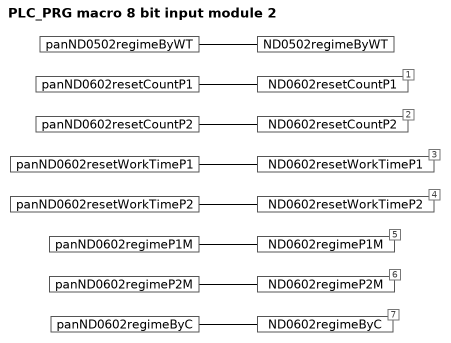
[picture p72: PLC_PRG macro 8 bit input module 2 (CFC)]
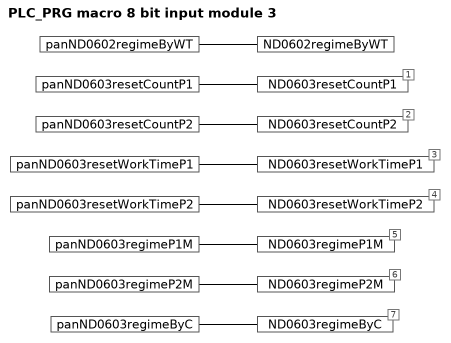
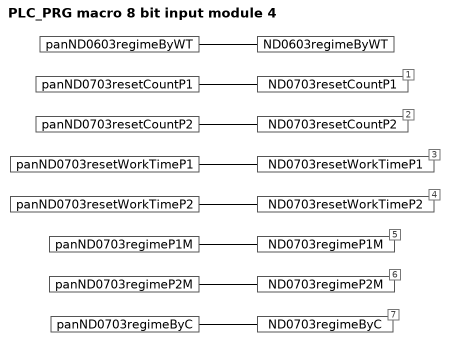
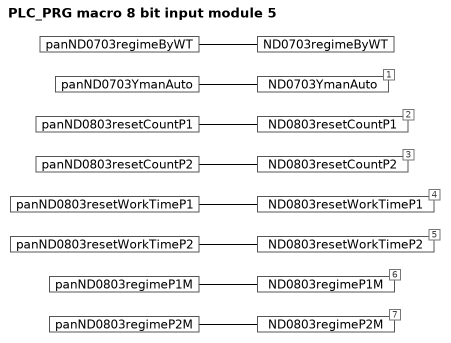
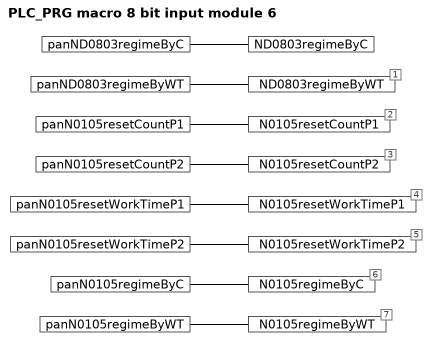
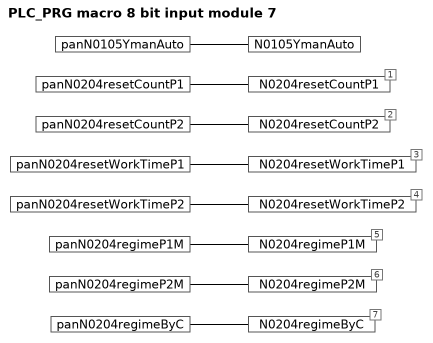
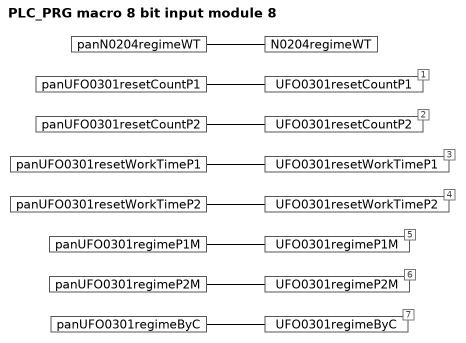
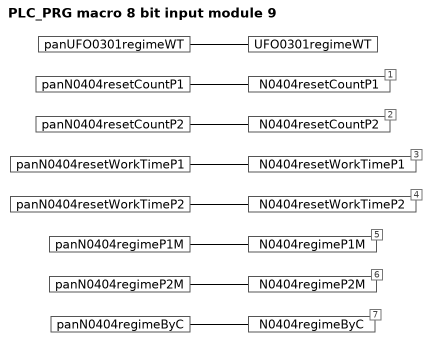
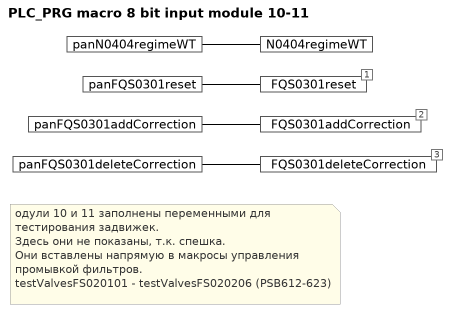
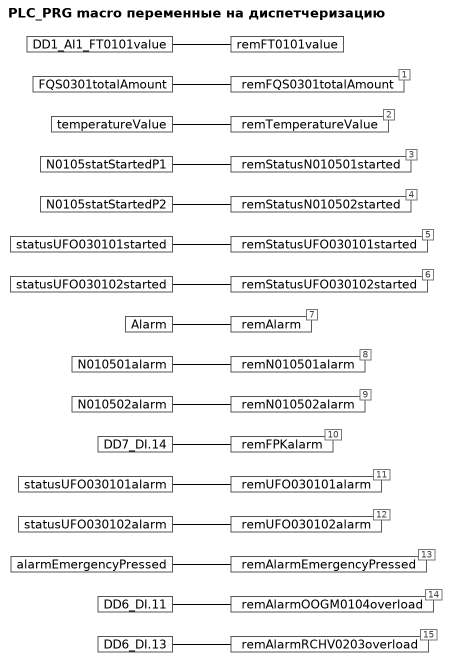
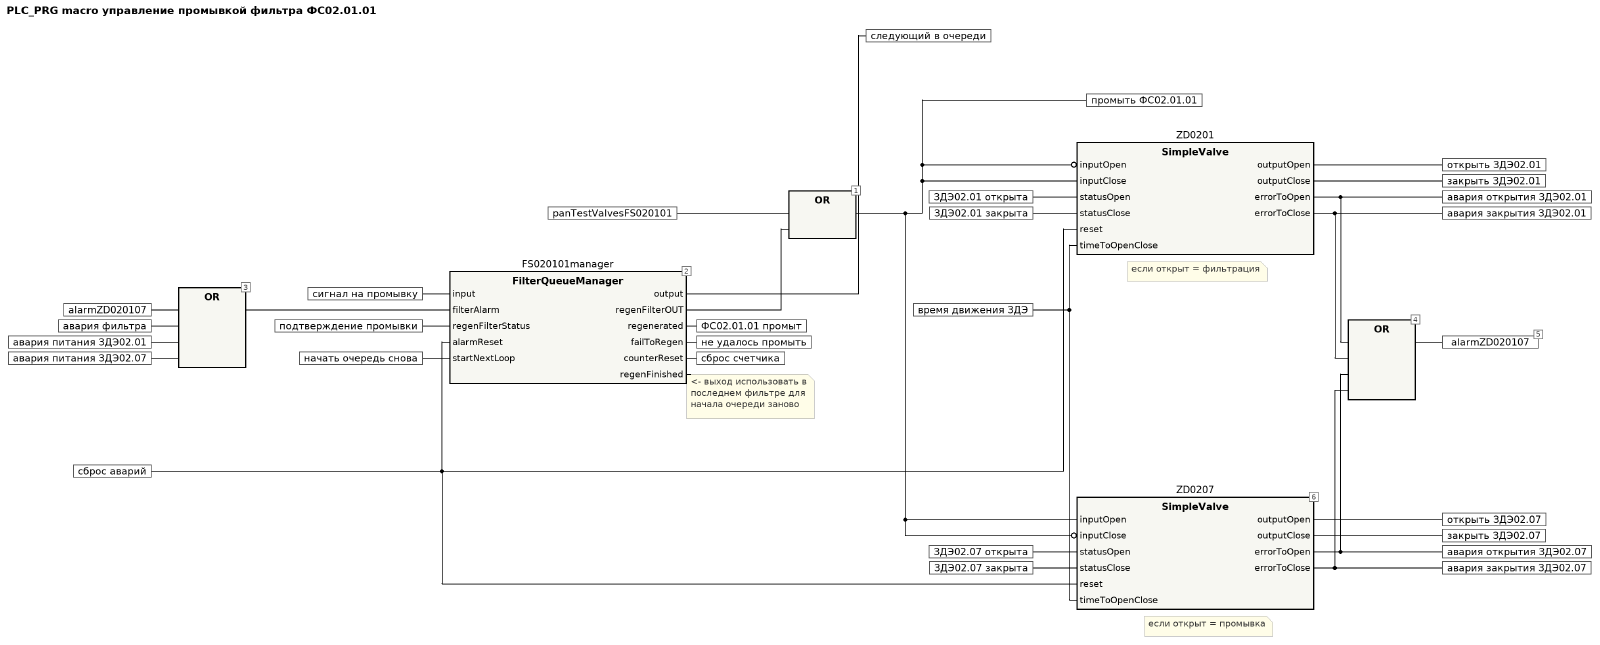
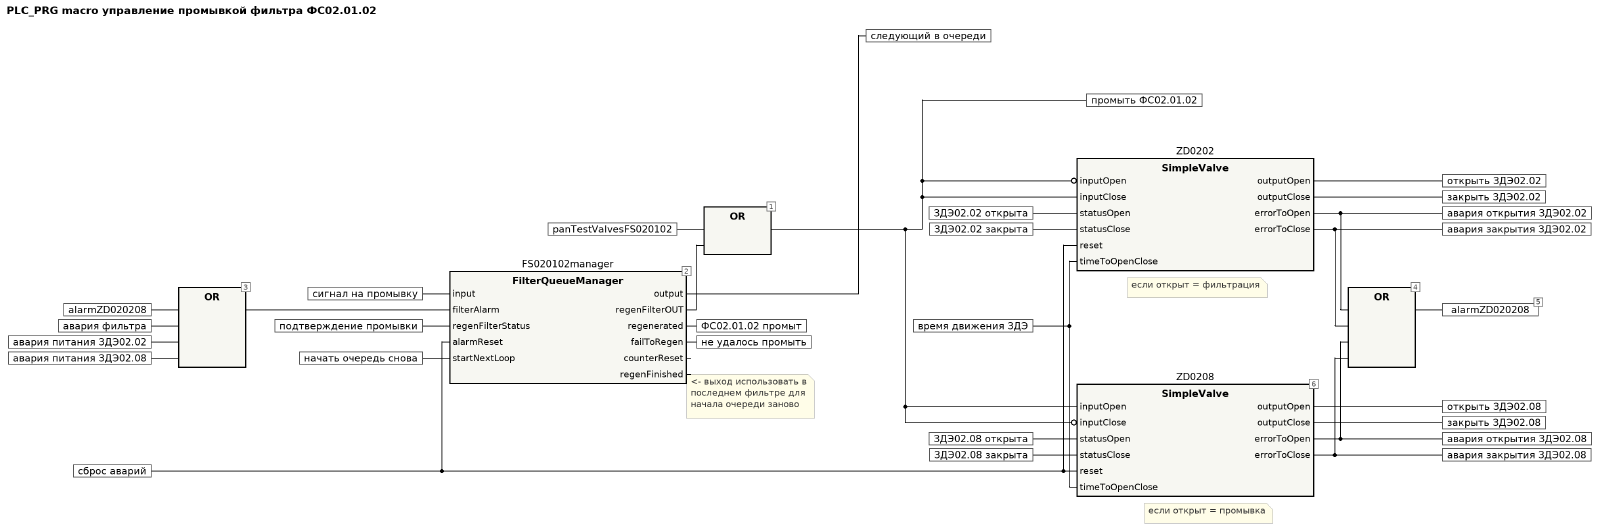
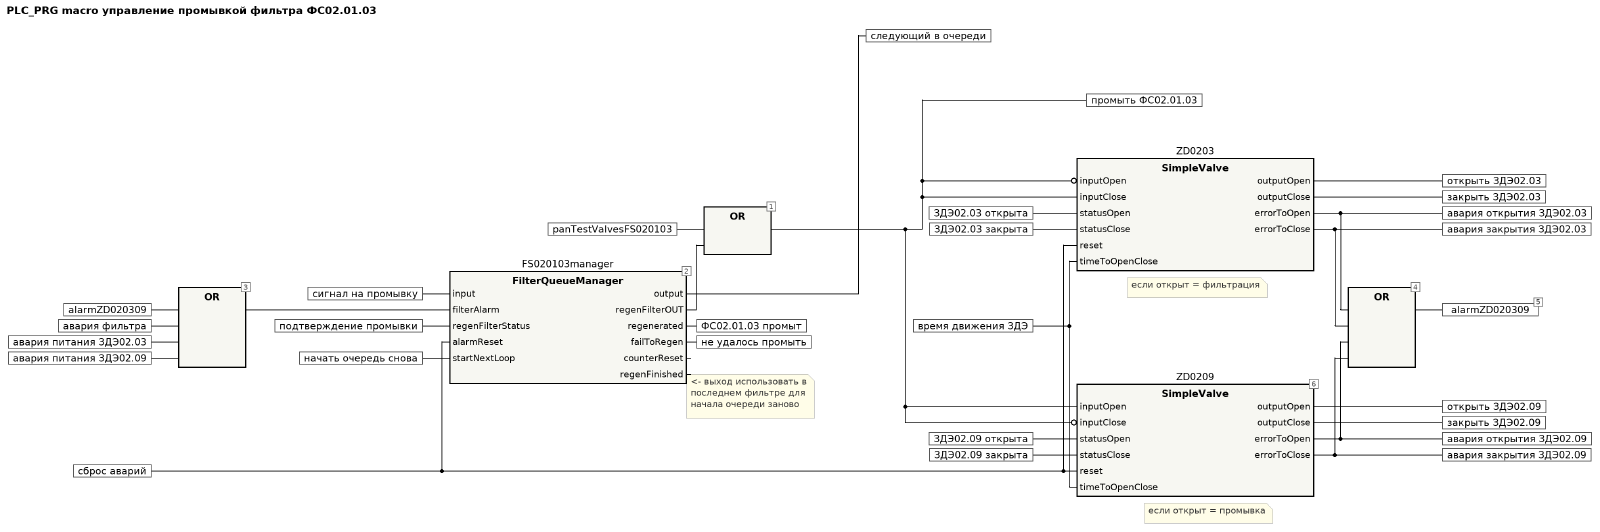
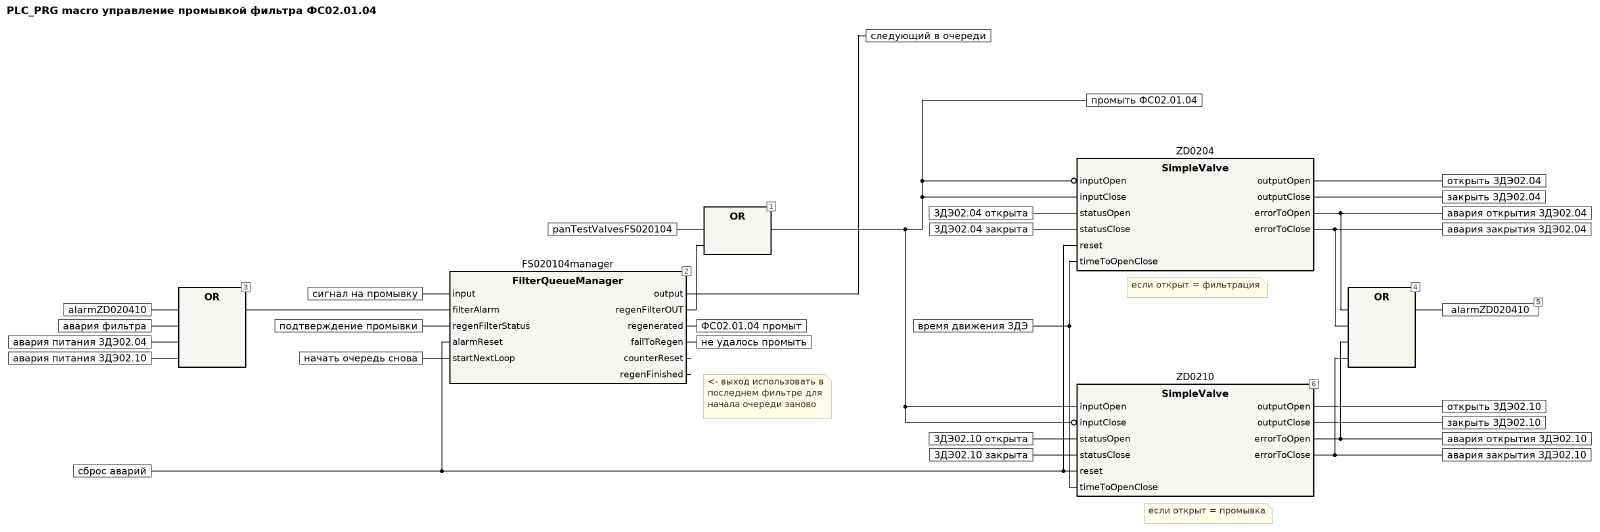
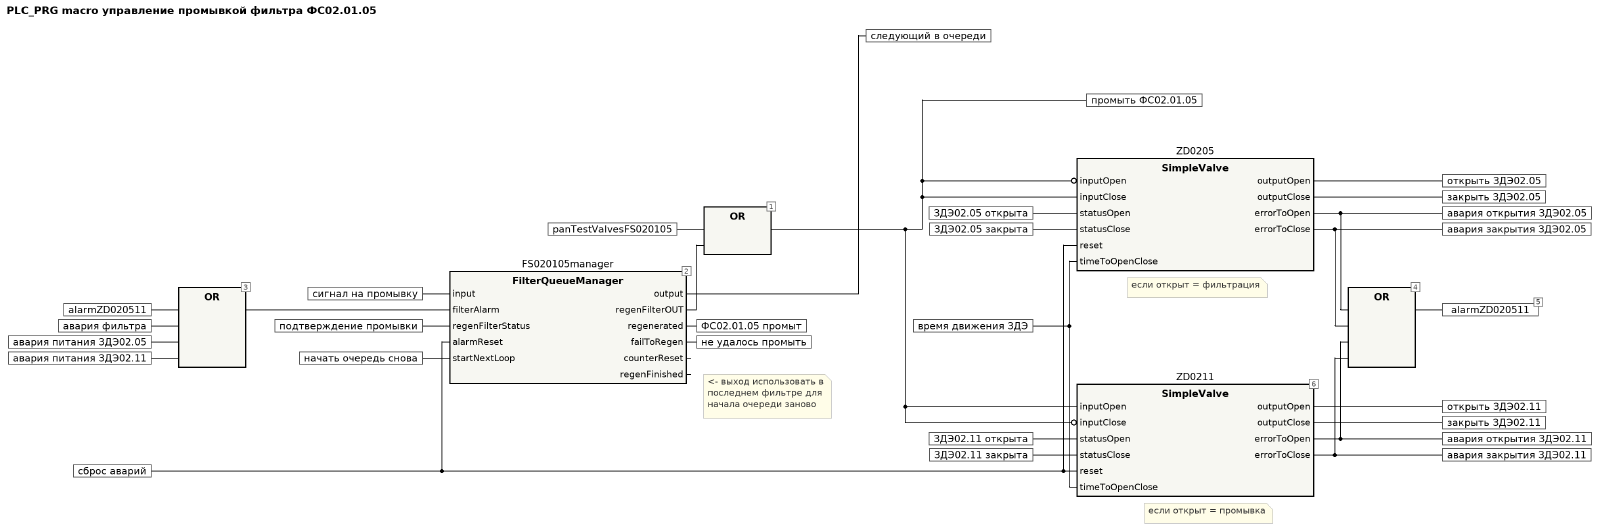
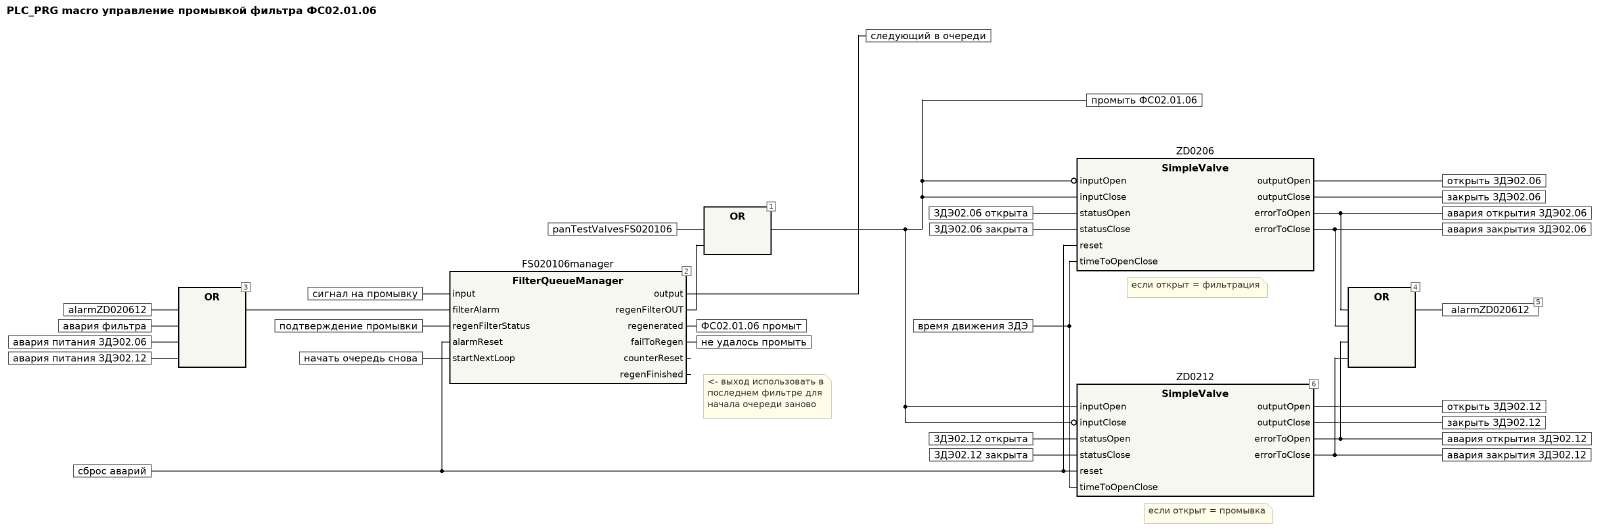
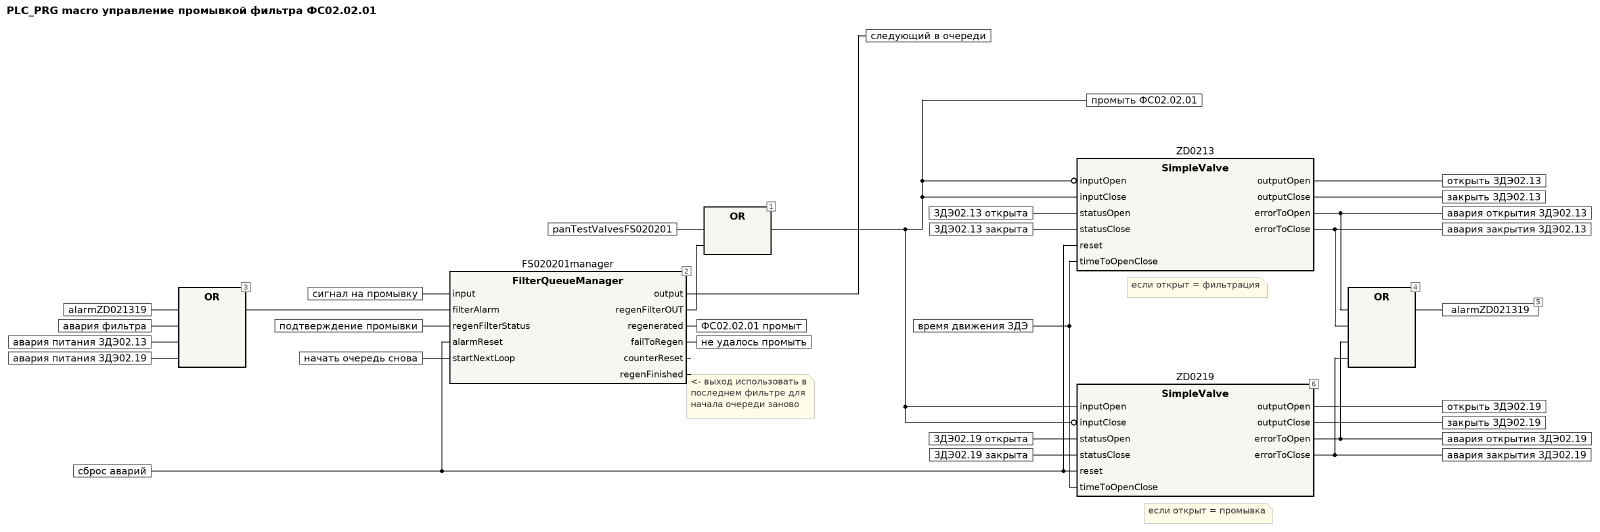
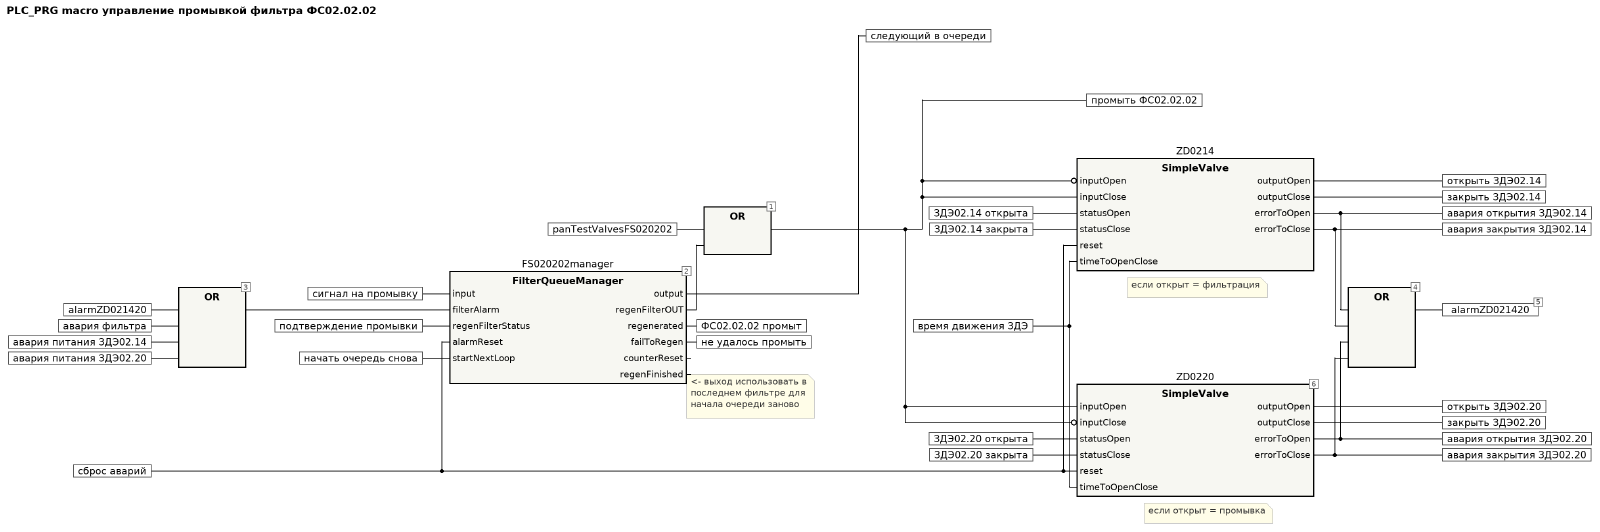
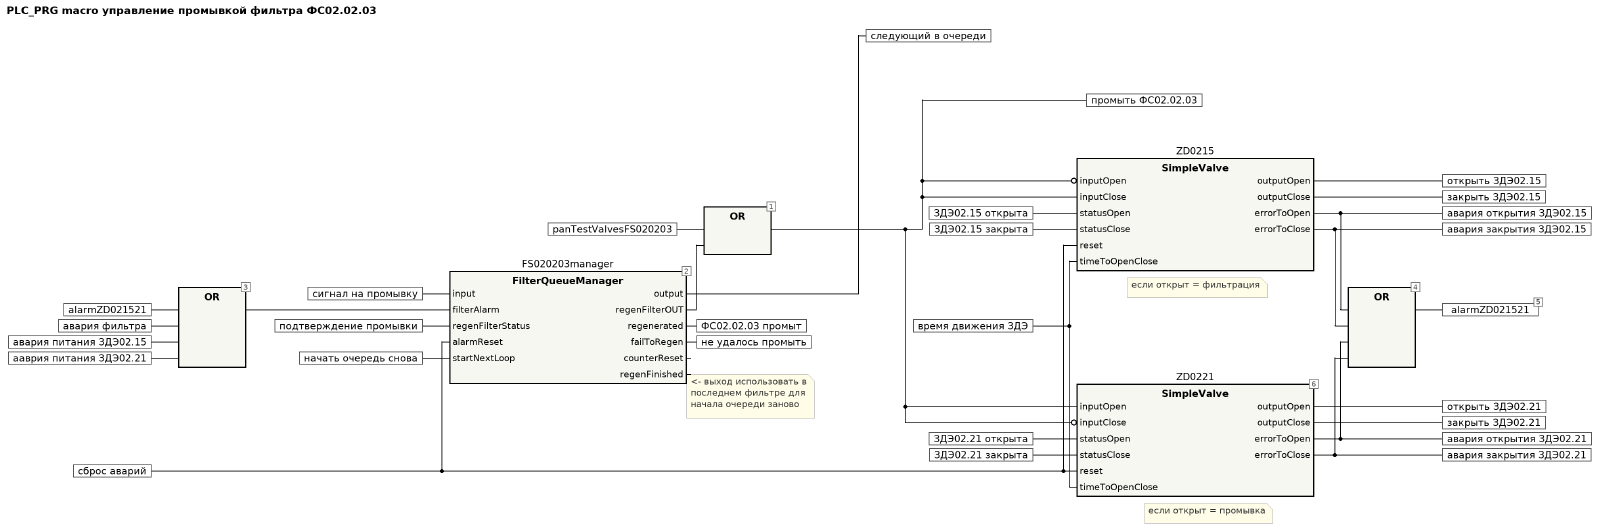
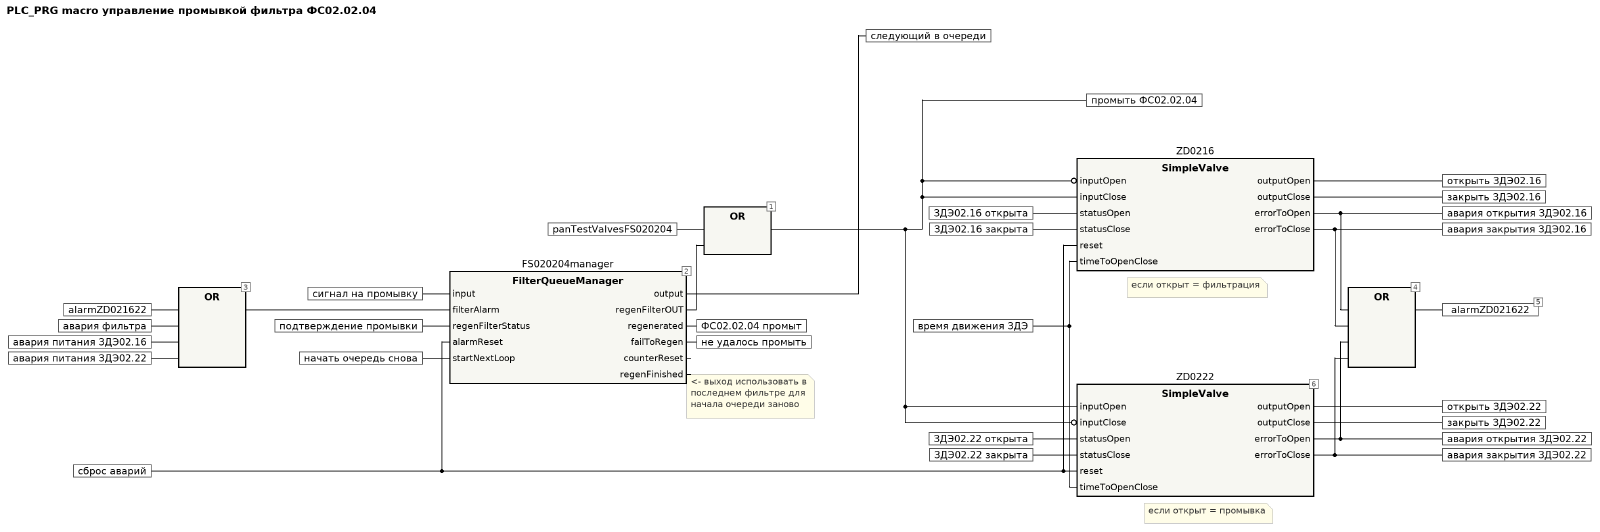
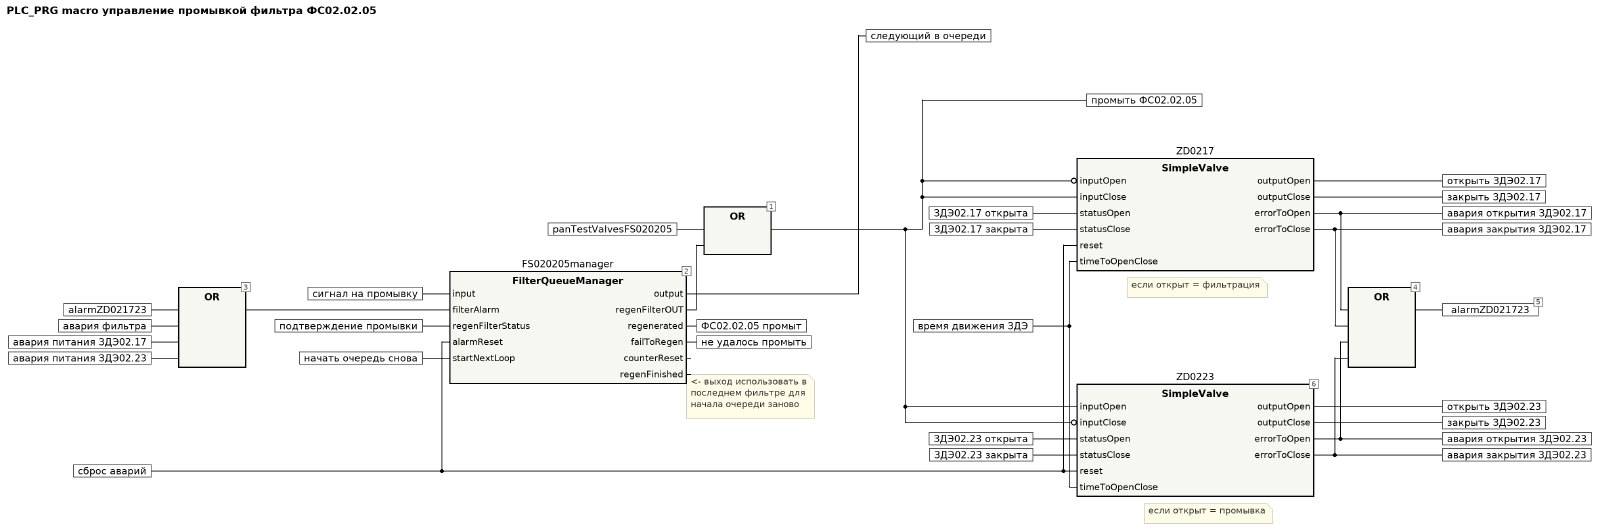
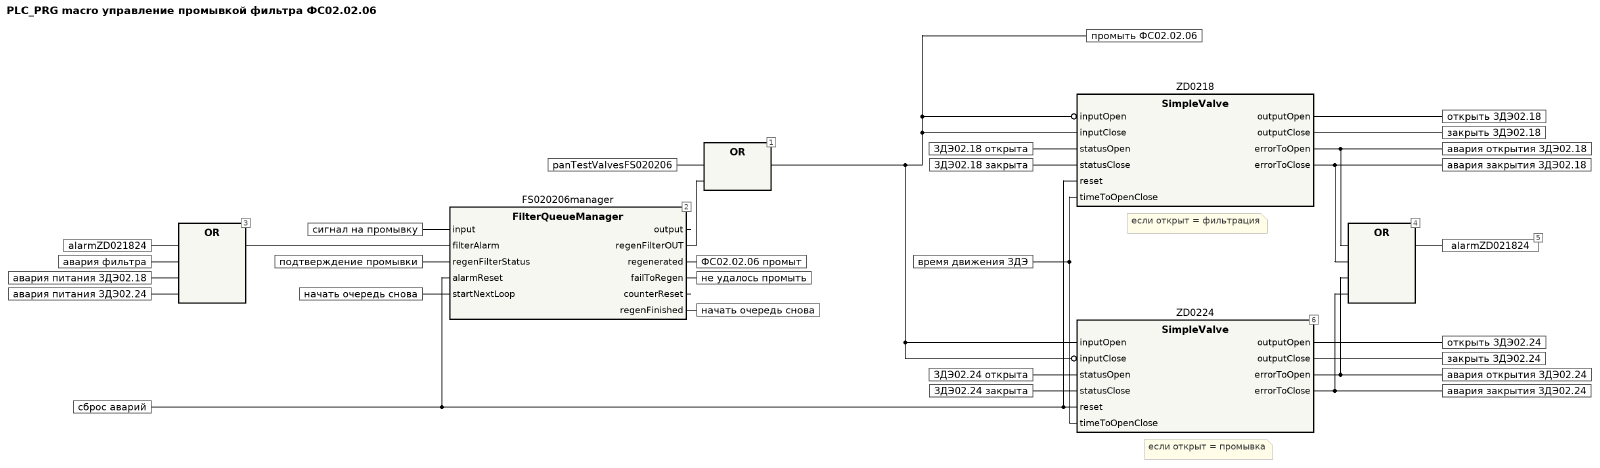
_CFC_ (* Continuous Function Chart, elements in execution order *)
(* 0 = перелив *)
(* авария обоих УФО, если проблемы / открытия/закрытия на одной из задвижек *)
(* авария питания ЗДЭ03.02 *)
(* авария питания ЗДЭ03.01 *)
(* статус-пуск Н01.05/02 *)
(* вкл КМ3 *)
(* Статус ПУСК / ЧРП Н01.05 *)
(* статус-пуск Н01.05/01 *)
(* вкл КМ2 *)
(* контроль обрыва или ошибок модулей в сети ПЛК *)
(* LSA01.02 перелив ОГМ01.04 *)
(* Нажат аварийный стоп. *)
(* авария сети (РКФ) *)
(* разрешение работы КНС / 1 = разрешено *)
(* Нажат аварийный стоп. *)
(* Блок управления разрешением работы КНС *)
(* авария сети (РКФ) *)
(* Авария питания клапанов КЭМ. *)
(* Авария питания розеток / управл.клапанов фильтров. *)
(* авария КНС *)
(* блок подачи сигнала на промывку *)
(* суммируем каждую секунду значение / мгновенного расхода в кубометрах в секунду *)
(* преобразуем расход из / кубометров в час в / кубометры в секунду *)
(* если есть расход / (больше нуля) *)
(* выдает импульс / каждую секунду *)
(* здесь мгновенный расход / в кубометрах в час (FT01.02) *)
(* Авария Н02.04/01 (0=авария) *)
(* Авария Н02.04/02 (0=авария) *)
(* промывка ФС02.01/06 *)
(* промывка ФС02.01/05 *)
(* промывка ФС02.01/04 *)
(* промывка ФС02.01/03 *)
(* промывка ФС02.01/02 *)
(* промывка ФС02.01/01 *)
(* пуск/стоп НД08.03/01 *)
(* пуск/стоп НД08.03/02 *)
(* пуск/стоп НД06.03/01 *)
(* пуск/стоп НД06.03/02 *)
(* пуск/стоп НД06.02/01 *)
(* пуск/стоп НД06.02/02 *)
(* пуск/стоп НД08.04 *)
(* пуск/стоп НД07.03/01 *)
(* пуск/стоп НД07.03/02 *)
(* авария М08.02 (УПФ) *)
(* авария М07.02 (УПЩ) *)
(* авария М06.04 (УПК) *)
(* работа М08.02 (УПФ) *)
(* работа М07.02 (УПЩ) *)
(* работа М06.04 (УПК) *)
(* Контроль, если УФО включили вручную, / а потока при этом нет. *)
(* авария УФО03.01/02 *)
(* работа УФО03.01/02 *)
(* авария УФО03.01/01 *)
(* Для подачи предостережения на пульте / оператора (при необходимости), а также / сигнализации лампой АВАРИЯ. *)
(* работа УФО03.01/01 *)
(* авария УФО03.01/02 *)
(* авария УФО03.01/01 *)
(* авария Н04.04/01 *)
(* авария Н04.04/02 *)
(* время контроля старта ФПК (по умолч.=3мин) *)
(* время работы ФПК после спада сигнала датч.осадка *)
(* запуск фильтрации *)
(* Защита от сухого хода насоса ФПК *)
(* датчик уровня осадка *)
(* Давление на входе ФПК (0...16 бар) *)
(* авария ФПК *)
(* подающий насос ФПК работает *)
(* ФПК готов к приему *)
(* ФПК не запустился *)
(* рН-метр QE01.02 на входе, / диапазон 0...14 *)
(* авария входа рН-метра QE01.01 *)
(* авария входа расходомера FT01.02 *)
(* расходомер FT01.01 на входе, / диапазон 0...600куб/час *)
(* авария НД08.04 *)
(* управление 4...20мА НД08.03/01 *)
(* пуск/стоп НД08.03/01 *)
(* пуск/стоп НД08.03/02 *)
(* управление 4...20мА НД08.03/02 *)
(* авария привода НД08.03/01 *)
(* авария привода НД08.03/02 *)
(* авария НД07.03/01 *)
(* авария НД07.03/02 *)
(* управление 4...20мА НД07.03/01 *)
(* управление 4...20мА НД07.03/02 *)
(* пуск/стоп НД07.03/01 *)
(* пуск/стоп НД07.03/02 *)
(* авария НД07.03/01 *)
(* авария НД07.03/02 *)
(* авария НД06.03/01 *)
(* авария НД06.03/02 *)
(* авария НД06.02/01 *)
(* авария НД06.02/02 *)
(* управление 4...20мА НД06.03/01 *)
(* пуск/стоп НД06.03/01 *)
(* пуск/стоп НД06.03/02 *)
(* управление 4...20мА НД06.03/02 *)
(* авария НД06.03/01 *)
(* авария НД06.03/02 *)
(* управление 4...20мА НД06.02/01 *)
(* пуск/стоп НД06.02/01 *)
(* пуск/стоп НД06.02/02 *)
(* управление 4...20мА НД06.02/02 *)
(* авария НД06.02/01 *)
(* авария НД06.02/02 *)
(* ошибка блока дозирования НД05.02 *)
(* авария входа датчика температуры *)
(* лампа АВАРИЯ *)
(* датчик температуры в помещении / (метран) диапазон: 0...+100С *)
(* управление 4...20мА НД05.02/01 *)
(* пуск/стоп НД05.02/01 *)
(* авария НД05.02/01 *)
(* авария НД05.02/02 *)
(* пуск/стоп НД05.02/02 *)
(* управление 4...20мА НД05.02/02 *)
(* АВАРИИ *)
(* авария привода НД08.03/01 *)
(* авария привода НД08.03/02 *)
(* авария НД08.04 *)
(* насос Н04.01 работает *)
(* пуск/стоп НД08.04 *)
(* управление 4...20мА НД08.04 *)
(* авария входа расходомера FT01.01 *)
(* расходомер FT01.02 на входе, / диапазон 0...600куб/час *)
(* рН-метр QE01.01 на входе, / диапазон 0...14 *)
(* авария входа рН-метра QE01.02 *)
(* сухой ход НД08.03/01 *)
(* сухой ход НД08.03/02 *)
(* сухой ход НД08.03/01 *)
(* сухой ход НД08.03/02 *)
(* LSA01.02 перелив ОГМ01.04 *)
(* Инициализирует требуемые булевые переменные / в момент старта выполнения программы. *)
(* Статус ПУСК ЧРП Н01.05 *)
(* LS01.03 - рабочий верхний уровень ОГМ01.04 автоматический пуск 01.05 *)
(* LS01.04 - нижний уровень ОГМ01.04, сухой ход Н01.05 *)
(* SA1 Ручной выбор Н01.05/01 = главный *)
(* SA1 Ручной выбор Н01.05/02 = главный *)
(* Стоп  Н01.05 (сброс самоподхвата реле) *)
(* время на создание потока *)
(* Пуск  Н01.05 *)
(* КМ1 питание ЧРП *)
(* КМ2 питание насоса 1 *)
(* КМ3 питание насоса 2 *)
(* Авария ЧРП Н01.05 *)
(* термоконтакт Н01.05/01 *)
(* термоконтакт Н01.05/02 *)
(* авария питания ЗДЭ02.25 *)
(* LSА02.01 Перелив РЧВ02.03 *)
(* Давление на входе ФПК / 0...16 бар (мах допуст.10) *)
(* Авария входа AI6 ПЛК, давл.ФПК *)
(* авария ФПК *)
(* Открыть КШЭ04.01 *)
(* статус КШЭ04.01 открыт *)
(* Закрыть КШЭ04.01 *)
(* статус КШЭ04.01 закрыт *)
(* подающий насос ФПК работает *)
(* стоп Н04.04 *)
(* пуск Н04.04/02 *)
(* пуск Н04.04/01 *)
(* авт.пуск Н04.04 *)
(* сухой ход Н04.04, 0=защита *)
(* авария Н04.04/01, 0=авария *)
(* авария Н04.04/02, 0=авария *)
(* импульсный расходомер *)
(* Авария Н02.04/01 (0=авария) *)
(* Авария Н02.04/02 (0=авария) *)
(* промывка ФС02.02/06 *)
(* промывка ФС02.02/05 *)
(* промывка ФС02.02/04 *)
(* промывка ФС02.02/03 *)
(* промывка ФС02.02/02 *)
(* промывка ФС02.02/01 *)
(* Клапан КЭМ05.01 открыт. *)
(* Клапан КЭМ06.01 открыт. *)
(* Клапан КЭМ07.01 открыт. *)
(* Клапан КЭМ08.01 открыт. *)
(* Сухой ход Н02.04 (LS02.03) 0=сух.ход *)
(* Стоп Н02.04 *)
(* Пуск Н02.04/01 *)
(* Пуск Н02.04/02 *)
(* текущий объем *)
(* заданный до промывки объем *)
(* 0=авария *)
(* авария (при 0) ФС02.01/06 *)
(* авария (при 0) ФС02.01/05 *)
(* авария (при 0) ФС02.01/04 *)
(* авария (при 0) ФС02.01/03 *)
(* авария (при 0) ФС02.01/02 *)
(* авария (при 0) ФС02.01/01 *)
(* авария (при 0) ФС02.02/06 *)
(* авария (при 0) ФС02.02/05 *)
(* авария (при 0) ФС02.02/04 *)
(* авария (при 0) ФС02.02/03 *)
(* авария (при 0) ФС02.02/02 *)
(* авария (при 0) ФС02.02/01 *)
(* сброс счетчика стоков до следующей промывки *)
(* подсчет общего объема стоков, прошедшего через расходомер FT01.02 *)
(* очередь передается на 2 ступень *)
(* авария питания ЗДЭ02.01 *)
(* авария питания ЗДЭ02.02 *)
(* авария питания ЗДЭ02.03 *)
(* авария питания ЗДЭ02.04 *)
(* авария питания ЗДЭ02.05 *)
(* авария питания ЗДЭ02.06 *)
(* авария питания ЗДЭ02.07 *)
(* авария питания ЗДЭ02.08 *)
(* авария питания ЗДЭ02.09 *)
(* авария питания ЗДЭ02.10 *)
(* авария питания ЗДЭ02.11 *)
(* авария питания ЗДЭ02.12 *)
(* авария питания ЗДЭ02.13 *)
(* авария питания ЗДЭ02.14 *)
(* авария питания ЗДЭ02.15 *)
(* авария питания ЗДЭ02.16 *)
(* авария питания ЗДЭ02.17 *)
(* авария питания ЗДЭ02.18 *)
(* авария питания ЗДЭ02.19 *)
(* авария питания ЗДЭ02.20 *)
(* авария питания ЗДЭ02.21 *)
(* авария питания ЗДЭ02.22 *)
(* авария питания ЗДЭ02.23 *)
(* авария питания ЗДЭ02.24 *)
(* инвертирование сигнала, чтобы все аварии / обозначались как 1 (TRUE) *)
(* авария НД05.02/01 *)
(* авария НД05.02/02 *)
(* авария питания КШЭ04.01 *)
(* 1=открыть; 0 = закрыть *)
(* в этом макросе лежит управление режимом тестирования задвижек ЗДЭ03 / Тестирование запрещает автоматический запуск УФО от ПЛК *)
#0 rTrigStartInitializer:R_TRIG(CLK: TRUE)
#1 startInitializer <= #0.Q
#2 MACRO контроль температуры в помещении(pin 1 "вход датчика температуры": DD1_AI0, pin 2 "минимально допустимая температура в помещении": maxTemperature, pin 3 "максимально допустимая температура в помещении": minTemperature)
	(* задаем границы допустимой температуры в помещении / проверяем что измеренное значение в заданном диапазоне *)
	(* не смотрим конкретный тип ошибки / (работает не точно, обрыв определяет как слишком маленькое значение) / если не равно 0 - значит на входе ошибка *)
	#3 DD1_AI0_temperature:DECODE_FLOAT(VALUE: pin 1, DEF_VALUE: -)
	#4 NE(#3._ERR, 0)
	out 2 "авария датчика температуры" <= #4
	out 1 "температура в помещении" <= #3.OUT_VALUE
	#5 REAL_TO_INT(#3.OUT_VALUE)
	#6 temperatureLimits:LIMITALARM(IN: #5, HIGH: pin 3, LOW: pin 2)
	out 3 "температура выше заданного диапазона" <= #6.O
	out 4 "температура ниже заданного диапазона" <= #6.U
	#7 temperatureLimits:LIMITALARM(IN: -, HIGH: -, LOW: -)
END_MACRO
#8 temperatureValue <= #2.out 1
#9 DD1_AI0_error <= #2.out 2
#10 alarmHighTemperature <= #2.out 3
#11 alarmLowTemperature <= #2.out 4
#12 OR(testKSHE0401, DD7_DI.13)
#13 MACRO клапан шаровый перед ФПК (КШЭ04.01)(pin 1 "сигнал "подающий насос ФПК" работает": #12, pin 2 "статус КШЭ04.01 открыт": DD9_DI.2, pin 3 "статус КШЭ04.01 закрыт": DD9_DI.3, pin 4 "сброс аварий": alarmReset, pin 5 "время на открытие/закрытие": timeToOpenCloseValve)
	#14 FPKkshe0401DelayToOpen:TON(IN: #16.outputOpen, PT: T#1s)
	out 1 "выход на открытие КШЭ04.01" <= #14.Q
	#15 FPKkshe0401DelayToClose:TON(IN: #16.outputClose, PT: T#1s)
	out 2 "выход на закрытие КШЭ04.01" <= #15.Q
	#16 FPKkshe0401:SimpleValve(inputOpen: pin 1, inputClose: #17, statusOpen: pin 2, statusClose: pin 3, reset: pin 4, timeToOpenClose: pin 5)
	#17 NOT(pin 1)
	out 3 "авария на открытие КШЭ04.01" <= #16.errorToOpen
	out 4 "авария на закрытие КШЭ04.01" <= #16.errorToClose
END_MACRO
#18 DD4_DO.2 <= #13.out 1
#19 DD4_DO.3 <= #13.out 2
#20 FPKkshe0401errorToOpen <= #13.out 3
#21 FPKkshe0401errorToClose <= #13.out 4
#22 OR(DD1_AI0_error, DD1_AI1_error, DD1_AI2_error, DD1_AI3_error, DD1_AI4_error, alarmHighTemperature, alarmLowTemperature, ND0502dosingError, ND0602dosingError, ND0603dosingError, ND0803dosingError, ND0804dosingError, DD1_DI6, DD1_DI7, N010501alarm, N010502alarm, ZDE0225errorToOpen, ZDE0225errorToClose, DD7_DI.14, FPKnotStarted, DD1_AI5_error, FPKkshe0401errorToOpen, FPKkshe0401errorToClose, DD5_DI.27, DD5_DI.29, filterFailToRegen020101, errorToOpenZD0201, errorToCloseZD0201, errorToOpenZD0207, errorToCloseZD0207, filterFailToRegen020102, errorToOpenZD0202, errorToCloseZD0202, errorToOpenZD0208, errorToCloseZD0208, filterFailToRegen020103, errorToOpenZD0203, errorToCloseZD0203, errorToOpenZD0209, errorToCloseZD0209, filterFailToRegen020104, errorToOpenZD0204, errorToCloseZD0204, errorToOpenZD0210, errorToCloseZD0210, filterFailToRegen020105, errorToOpenZD0205, errorToCloseZD0205, errorToOpenZD0211, errorToCloseZD0211, filterFailToRegen020106, errorToOpenZD0206, errorToCloseZD0206, errorToOpenZD0212, errorToCloseZD0212, filterFailToRegen020201, errorToOpenZD0213, errorToCloseZD0213, errorToOpenZD0219, errorToCloseZD0219, filterFailToRegen020202, errorToOpenZD0214, errorToCloseZD0214, errorToOpenZD0220, errorToCloseZD0220, filterFailToRegen020203, errorToOpenZD0215, errorToCloseZD0215, errorToOpenZD0221, errorToCloseZD0221, filterFailToRegen020204, errorToOpenZD0216, errorToCloseZD0216, errorToOpenZD0222, errorToCloseZD0222, filterFailToRegen020205, errorToOpenZD0217, errorToCloseZD0217, errorToOpenZD0223, errorToCloseZD0223, filterFailToRegen020206, errorToOpenZD0218, errorToCloseZD0218, errorToOpenZD0224, errorToCloseZD0224, alarmPLKnetwork, alarmND050201, alarmND050202, alarmND060201, alarmND060202, alarmND060301, alarmND060302, alarmND070301, alarmND070302, alarmND080301, alarmND080302, alarmND0804, alarmOGM0104overload, alarmRCHV0203overload, alarmN040402, alarmN040401, alarmM0604, alarmM0702, alarmM0802, alarmN020401, alarmN020402, alarmFS020101, alarmFS020102, alarmFS020103, alarmFS020104, alarmFS020105, alarmFS020106, alarmFS020201, alarmFS020202, alarmFS020203, alarmFS020204, alarmFS020205, alarmFS020206, alarmZDE0201power, alarmZDE0202power, alarmZDE0203power, alarmZDE0204power, alarmZDE0205power, alarmZDE0206power, alarmZDE0207power, alarmZDE0208power, alarmZDE0209power, alarmZDE0210power, alarmZDE0211power, alarmZDE0212power, alarmZDE0213power, alarmZDE0214power, alarmZDE0215power, alarmZDE0216power, alarmZDE0217power, alarmZDE0218power, alarmZDE0219power, alarmZDE0220power, alarmZDE0221power, alarmZDE0222power, alarmZDE0223power, alarmZDE0224power, alarmZDE0225power, alarmKSHE0401power, alarmKNS, alarmPowerSocketFS, alarmKEMvalvesPower, alarmEmergencyPressed, alarmRKF, errorToOpenZDE0301, errorToCloseZDE0301, errorToOpenZDE0302, errorToCloseZDE0302, alarmZDE0301power, alarmZDE0302power)
#23 DD1_DO11 <= #22
#24 alarm <= #22
#25 MACRO контроль аналогового входа DD1_AI1(pin 1 "вход": DD1_AI1)
	(* Не смотрим конкретную ошибку, / определяем,что вход неисправен без расшифровки. *)
	#26 DD1_AI1_FT0101:DECODE_FLOAT(VALUE: pin 1, DEF_VALUE: -)
	#27 NE(#26._ERR, 0)
	out 2 "авария" <= #27
	out 1 "выход" <= #26.OUT_VALUE
END_MACRO
#28 DD1_AI1_FT0101value <= #25.out 1
#29 DD1_AI1_error <= #25.out 2
#30 MACRO контроль аналогового входа DD1_AI2(pin 1 "вход": DD1_AI2)
	(* Не смотрим конкретную ошибку, / определяем,что вход неисправен без расшифровки. *)
	#31 DD1_AI2_FT0102:DECODE_FLOAT(VALUE: pin 1, DEF_VALUE: -)
	#32 NE(#31._ERR, 0)
	out 2 "авария" <= #32
	out 1 "выход" <= #31.OUT_VALUE
END_MACRO
#33 DD1_AI2_FT0102value <= #30.out 1
#34 DD1_AI2_error <= #30.out 2
#35 MACRO управление Н01.05 (поддержание заданного расхода по FT01.02)(pin 1 "статус ПУСК ЧРП (реле)": DD5_DI.4, pin 2 "LS01.03 раб.уров.": DD6_DI.12, pin 3 "LS01.04 ниж.уров.(сух.ход)": DD5_DI.0, pin 4 "SA1ручной выб.Н01.05/01-главный": DD5_DI.5, pin 5 "SA1ручной выб.Н01.05/02-главный": DD5_DI.6, pin 6 "включить режим "по кол.вкл."": N0105regimeByC, pin 7 "включить режим "по наработке"": N0105regimeByWT, pin 8 "значение расхода от FT01.02": DD1_AI2_FT0102value, pin 9 "уставка расхода": N0105flowSetValue, pin 10 "время на создание потока": N0105minFlowTime, pin 11 "Р-коэфф.": N0105koeffP, pin 12 "I-коэфф": N0105koeffI, pin 13 "Д-коэфф": N0105koeffD, pin 14 "управление ЧРП в ручн.реж.(4...20мА)": N0105YoutManual, pin 15 "переключатель управление ЧРП РУЧН/АВТ": N0105YmanAuto, pin 16 "мин.допустимый расход": N0105minFlow, pin 17 "термоконтакт Н01.05/01": DD5_DI.2, pin 18 "термоконтакт Н01.05/02": DD5_DI.3, pin 19 "авария ЧРП Н01.05": DD5_DI.1, pin 20 "сброс аварии": alarmReset, pin 21 "сброс кол-ва вкл.Н01.05/01": N0105resetCountP1, pin 22 "сброс кол-ва вкл.Н01.05/02": N0105resetCountP2, pin 23 "сброс наработки Н01.05/01": N0105resetWorkTimeP1, pin 24 "сброс наработки Н01.05/02": N0105resetWorkTimeP2)
	(* время на создание потока *)
	(* Пуск  Н01.05 *)
	(* режимы по количеству включений,  или по наработке / активны если оба входа SA1 не активны *)
	(* управление Н01.05 - поддержание / заданного расхода по FT01.02 *)
	(* по умолчанию при старте программы *)
	(* если на входе true / то нижнее значение, / иначе то, что посередине *)
	(* Если насос создает давление меньше / указанного, то авария. *)
	#36 OR(pin 2, #37.Q)
	#37 N0105startTrig:R_TRIG(CLK: pin 1)
	#38 N0105stopTrig:F_TRIG(CLK: pin 1)
	#39 N0105startTrigg:RS(SET: #36, RESET1: #41)
	#40 N0105regime:choosePumpRegime(start: #39.Q1, pump1Main: pin 4, pump2Main: pin 5, byCounter: #44, byWorkTime: #50)
	out 2 "статус режим "Н01.05/01 - главный"" <= #40.pump1MainActive
	out 3 "статус режим "Н01.05/02 - главный"" <= #40.pump2MainActive
	out 4 "статус режим "по кол-ву вкл."" <= #40.byCounterActive
	#41 OR(#38.Q, #42)
	out 5 "статус режим "по наработке"." <= #40.byWorkTimeActive
	#42 NOT(pin 3)
	#43 NOT(#39.Q1)
	out 1 "СТОП (сброс самоподхвата реле пуска ЧРП)." <= #43
	#44 AND(NOT pin 4, NOT pin 5, #47.Q1)
	#45 OR(pin 6, startInitializer)
	#46 N0105regByCinit:R_TRIG(CLK: #45)
	#47 N0105regByCtrig:RS(SET: #46.Q, RESET1: #55.Q)
	#48 N0105twoPumpOneDriveManager:TwoPumpOneDriveManager(startStopPump1: #40.startPump1, startStopPump2: #40.startPump2, alarmPump1: N010501alarm, alarmPump2: N010502alarm, alarmReset: alarmReset, counterStart: #40.startByCounter, Pump1ResetCounter: pin 21, Pump2ResetCounter: pin 22, ValueToResetCounter: -, workTimeStart: #40.startByWorkTime, workTimePump1Reset: pin 23, workTimePump2Reset: pin 24, timeKM1off: -, timeKM23DelayON: -, timeKM23offDelay: -, timeReadyToStartDelay: -)
	out 6 "кол-во включений Н01.05/01" <= #48.counterPump1
	#49 AND(#48.pump1active, #65)
	out 7 "кол-во включений Н01.05/02" <= #48.counterPump2
	out 8 "наработка Н01.05/01" <= #48.currentWorkTimePump1
	out 15 "авария Н01.05/01" <= #53.Q1
	#50 AND(NOT pin 4, NOT pin 5, #56.Q1)
	out 9 "наработка Н01.05/02" <= #48.currentWorkTimePump2
	out 10 "КМ1-питание ЧРП" <= #48.DriveKM
	#51 AND(#48.pump1active, #57)
	#52 OR(#49, #51)
	#53 N010501alarmTrig:RS(SET: #52, RESET1: pin 20)
	#54 N010501alarm <= #53.Q1
	#55 N0105regWTinit:R_TRIG(CLK: pin 7)
	#56 N0105regWTtrig:RS(SET: #55.Q, RESET1: #46.Q)
	out 11 "КМ2-питание Н01.05/01" <= #48.pump1KM
	out 12 "КМ3-питание Н01.05/02" <= #48.pump2KM
	#57 OR(NOT pin 17, NOT pin 19)
	out 13 "пуск ЧРП (Н01.05)" <= #48.driveStart
	#58 OR(NOT pin 19, NOT pin 18)
	out 16 "авария Н01.05/02" <= #61.Q1
	#59 AND(#58, #48.pump2active)
	#60 OR(#59, #63)
	#61 N010502alarmTrig:RS(SET: #60, RESET1: pin 20)
	#62 N010502alarm <= #61.Q1
	#63 AND(#48.pump2active, #65)
	#64 N0105timerminFlow:TON(IN: #48.driveStart, PT: pin 10)
	#65 AND(#64.Q, #66)
	#66 LE(pin 8, pin 16)
	#67 SEL(#48.driveStart, 0, #68.Y)
	out 14 "управление ЧРП (4...20мА)" <= #67
	#68 N0105pidReg:PID(ACTUAL: pin 8, SET_POINT: pin 9, KP: pin 11, TN: pin 12, TV: pin 13, Y_MANUAL: pin 14, Y_OFFSET: -, Y_MIN: 4, Y_MAX: 20, MANUAL: pin 15, RESET: #68.OVERFLOW)
END_MACRO
#69 DD4_DO.13 <= #35.out 1
#70 N0105statRegimeP1M <= #35.out 2
#71 N0105statRegimeP2M <= #35.out 3
#72 N0105statRegimeByC <= #35.out 4
#73 N0105statRegimeByWT <= #35.out 5
#74 N0105counterP1 <= #35.out 6
#75 N0105counterP2 <= #35.out 7
#76 N0105workTimeP1 <= #35.out 8
#77 N0105workTimeP2 <= #35.out 9
#78 DD2_DO.0 <= #35.out 10
#79 DD2_DO.1 <= #35.out 11
#80 DD2_DO.2 <= #35.out 12
#81 DD1_DO0 <= #35.out 13
#82 DD1_AO0 <= #35.out 14
#83 N010501alarm <= #35.out 15
#84 N010502alarm <= #35.out 16
#85 MACRO Сигналы работы с ФП04.02 (фильтр-пресс)(pin 1 "датчик уровня осадка": DD7_DI.15, pin 2 "время работы ФПК (после выкл.датч.осадка)": FPKtimeToWork, pin 3 "защита от сухого хода": DD6_DI.10, pin 4 "ошибка входа AI (обрыв)": DD1_AI5_error, pin 5 "авария ФПК": DD7_DI.14, pin 6 "фильтр-пресс готов к приему": DD7_DI.12, pin 7 "давление на входе в ФПК": DD1_AI5_FPKpressureValue, pin 8 "мах допустимое давление": FPKmaxPressureValue, pin 9 "подающий насос ФПК работает": DD7_DI.13, pin 10 "время контроля старта ФПК": FPKnotStartedTime, pin 11 "сброс аварий": alarmReset)
	(* ФПК готов к приему осадка *)
	(* LS01.01-нижн.уровень на входе ОГМ01.04 / защита от сух. хода насоса ФПК *)
	(* LES01.01-сигнал датчика уровня осадка ОГМ01.04 / запуск процесса фильтрации *)
	(* Время работы ФПК после / спада сигнала уровня осадка / по умолч.15мин. *)
	(* Давление на входе ФПК / 0...16 бар (мах допуст.10) *)
	(* максимально допустимое давление / на входе ФПК *)
	(* Условие сброса сигнала о грязном фильтр-прессе: / 1. Пропал сигнал о готовности ФПК; / 2. Появился сигнал о готовности ФПК. / Это значит, что оператор раздвигал плиты, / чистил и снова сдвигал их. *)
	#86 FPKneedToCleanResetFtrig:F_TRIG(CLK: FPKneedToCleanReset)
	#87 FPKstartTrig:RS(SET: pin 1, RESET1: #93)
	out 1 "запуск/старт ФПК" <= #87.Q1
	#88 FPKstopTimer:TOF(IN: pin 1, PT: pin 2)
	#89 FPKstopFtrig:F_TRIG(CLK: #88.Q)
	#90 AND(#87.Q1, #91)
	#91 NOT(pin 11)
	#92 AND(#87.Q1, #94.Q, #96)
	out 2 "ФПК не стартовал" <= #92
	#93 OR(#89.Q, pin 4, pin 5, #95, #97, #100.Q1)
	#94 FPKnotStartedTimer:TON(IN: #90, PT: pin 10)
	#95 NOT(pin 3)
	#96 NOT(pin 9)
	#97 NOT(pin 6)
	#98 AND(#87.Q1, #99)
	#99 GE(pin 7, pin 8)
	#100 FPKneedToCleanTrig:RS(SET: #98, RESET1: #86.Q)
	out 3 "ФПК нужно почистить!" <= #100.Q1
	#101 S FPKneedToCleanReset <= #100.Q1
	#102 FPKneedToCleanResetRtrig:R_TRIG(CLK: pin 6)
	#103 R FPKneedToCleanReset <= #102.Q
END_MACRO
#104 DD1_DO10 <= #85.out 1
#105 FPKnotStarted <= #85.out 2
#106 FPKneedToClean <= #85.out 3
#107 MACRO контроль аналогового входа DD1_AI3(pin 1 "вход": DD1_AI3)
	(* Не смотрим конкретную ошибку, / определяем,что вход неисправен без расшифровки. *)
	#108 DD1_AI3_QE0101:DECODE_FLOAT(VALUE: pin 1, DEF_VALUE: -)
	#109 NE(#108._ERR, 0)
	out 2 "авария" <= #109
	out 1 "выход" <= #108.OUT_VALUE
END_MACRO
#110 DD1_AI3_QE0101value <= #107.out 1
#111 DD1_AI3_error <= #107.out 2
#112 MACRO контроль аналогового входа DD1_AI4(pin 1 "вход": DD1_AI4)
	(* Не смотрим конкретную ошибку, / определяем,что вход неисправен без расшифровки. *)
	#113 DD1_AI4_QE0102:DECODE_FLOAT(VALUE: pin 1, DEF_VALUE: -)
	#114 NE(#113._ERR, 0)
	out 2 "авария" <= #114
	out 1 "выход" <= #113.OUT_VALUE
END_MACRO
#115 DD1_AI4_QE0102value <= #112.out 1
#116 DD1_AI4_error <= #112.out 2
#117 MACRO контроль аналогового входа DD1_AI5(pin 1 "вход": DD1_AI5)
	(* Не смотрим конкретную ошибку, / определяем,что вход неисправен без расшифровки. *)
	#118 DD1_AI5_FPK:DECODE_FLOAT(VALUE: pin 1, DEF_VALUE: -)
	#119 NE(#118._ERR, 0)
	out 2 "авария" <= #119
	out 1 "выход" <= #118.OUT_VALUE
END_MACRO
#120 DD1_AI5_FPKpressureValue <= #117.out 1
#121 DD1_AI5_error <= #117.out 2
#122 MACRO управление НД05.02 УПГ(pin 1 "вход расходомера в куб/час": DD1_AI1_FT0101value, pin 2 "max производительность НД в мл/мин": ND0502setMaxDosVal, pin 3 "задание дозирования в мл/куб": ND0502setKoefProp, pin 4 "режим:1 насос главный": ND0502regimeP1M, pin 5 "режим: 2 насос главный": ND0502regimeP2M, pin 6 "режим: по наработке": ND0502regimeByWT, pin 7 "режим: по кол-ву включений": ND0502regimeByC, pin 8 "авария 1 насоса": DD6_DI.0, pin 9 "авария 2 насоса": DD6_DI.1, pin 10 "сброс аварий": alarmReset, pin 11 "сброс счетчика включений 1 насоса": ND0502resetCountP1, pin 12 "сброс ссчетчика включений 2 насоса": ND0502resetCountP2, pin 13 "сброс наработки 1 насоса": ND0502resetWorkTimeP1, pin 14 "сброс наработки 2 насоса": ND0502resetWorkTimeP2)
	(* сигнал 4...20мА на НД05.02/02 *)
	(* сигнал 4...20мА на НД05.02/01 *)
	(* Если на входе SEL = TRUE, / то нижнее значение, / иначе - то,что посередине. *)
	#123 SEL(#129.pump1ON, 0, #124.outputValue)
	out 6 "выход 4...20мА насоса 1" <= #123
	#124 ND0502dosing:DosingPumpProportional(flowValue: pin 1, setMinPumpDosingValue: -, setMaxPumpDosingValue: pin 2, minOutputValue: -, maxOutputValue: -, setKoeffProportionality: pin 3, minFlowToStart: -)
	out 1 "ошибка блока дозирования" <= #124.dosingError
	#125 SEL(#129.pump2ON, 0, #124.outputValue)
	#126 REAL_TO_WORD(#125)
	out 7 "выход 4...20мА насоса 2" <= #126
	#127 ND0502regime:choosePumpRegime(start: #124.startDosingPump, pump1Main: pin 4, pump2Main: pin 5, byCounter: #128, byWorkTime: pin 6)
	out 2 "статус: 1 насос главный" <= #127.pump1MainActive
	out 3 "статус: 2 насос главный" <= #127.pump2MainActive
	out 4 "статус: по кол-ву включений" <= #127.byCounterActive
	#128 OR(pin 7, startInitializer)
	out 5 "статус: по наработке" <= #127.byWorkTimeActive
	#129 ND0502manager:TwoPumpManager(startStopPump1: #127.startPump1, startStopPump2: #127.startPump2, alarmPump1: #130, alarmPump2: #131, alarmReset: pin 10, counterStart: #127.startByCounter, Pump1ResetCounter: pin 11, Pump2ResetCounter: pin 12, ValueToResetCounter: -, workTimeStart: #127.startByWorkTime, workTimePump1Reset: pin 13, workTimePump2Reset: pin 14)
	out 12 "сигнал на включение насоса 1" <= #129.pump1ON
	#130 NOT(pin 8)
	out 13 "сигнал на включение насоса 2" <= #129.pump2ON
	out 8 "счетчик включений насоса 1" <= #129.counterPump1
	#131 NOT(pin 9)
	out 9 "счетчик включений насоса 2" <= #129.counterPump2
	out 10 "счетчик наработки насоса 1" <= #129.currentWorkTimePump1
	out 11 "счетчик наработки насоса 2" <= #129.currentWorkTimePump2
END_MACRO
#132 ND0502dosingError <= #122.out 1
#133 ND0502statRegimeP1M <= #122.out 2
#134 ND0502statRegimeP2M <= #122.out 3
#135 ND0502statRegimeByC <= #122.out 4
#136 ND0502statRegimeByWT <= #122.out 5
#137 DD1_AO3 <= #122.out 6
#138 DD10_AO0 <= #122.out 7
#139 ND0502counterP1 <= #122.out 8
#140 ND0502counterP2 <= #122.out 9
#141 ND0502workTimeP1 <= #122.out 10
#142 ND0502workTimeP2 <= #122.out 11
#143 DD4_DO.4 <= #122.out 12
#144 DD4_DO.5 <= #122.out 13
#145 AND(DD2_DO.1, DD5_DI.4)
#146 N0105statStartedP1 <= #145
#147 AND(DD5_DI.4, DD2_DO.2)
#148 N0105statStartedP2 <= #147
#149 MACRO Наполнение РЧВ02.03 (заслонка ЗДЭ02.25)(pin 1 "LS02.02раб.верх.уровень РЧВ": DD6_DI.14, pin 2 "LSA02.01 Перелив РЧВ": DD6_DI.13, pin 3 "статус ЗДЭ02.25 открыт": DD9_DI.0, pin 4 "статус ЗДЭ02.25 закрыт": DD9_DI.1, pin 5 "сброс аварий": alarmReset, pin 6 "время на открытие/закрытие": timeToOpenCloseValve)
	#150 OR(testZDE0225, pin 1)
	#151 NOT(pin 1)
	#152 ZDE0225:SimpleValve(inputOpen: #150, inputClose: #153, statusOpen: pin 3, statusClose: pin 4, reset: pin 5, timeToOpenClose: pin 6)
	out 1 "выход на открытие ЗДЭ02.25" <= #152.outputOpen
	#153 OR(#151, #154)
	out 2 "выход на закрытие ЗДЭ02.25" <= #152.outputClose
	out 3 "авария на открытие ЗДЭ02.25" <= #152.errorToOpen
	#154 NOT(pin 2)
	out 4 "авария на закрытие ЗДЭ02.25" <= #152.errorToClose
END_MACRO
#155 DD4_DO.0 <= #149.out 1
#156 DD4_DO.1 <= #149.out 2
#157 ZDE0225errorToOpen <= #149.out 3
#158 ZDE0225errorToClose <= #149.out 4
#159 MACRO управление Н02.04 (подача из РЧВ)(pin 1 "промывка ФС02.01/01": DD6_DI.20, pin 2 "промывка ФС02.01/02": DD6_DI.22, pin 3 "промывка ФС02.01/03": DD6_DI.24, pin 4 "промывка ФС02.01/04": DD6_DI.26, pin 5 "промывка ФС02.01/05": DD6_DI.28, pin 6 "промывка ФС02.01/06": DD6_DI.30, pin 7 "промывка ФС02.02/01": DD7_DI.0, pin 8 "промывка ФС02.02/02": DD7_DI.2, pin 9 "промывка ФС02.02/03": DD7_DI.4, pin 10 "промывка ФС02.02/04": DD7_DI.6, pin 11 "промывка ФС02.02/05": DD7_DI.8, pin 12 "промывка ФС02.02/06": DD7_DI.10, pin 13 "открыт КЭМ05.01": DD1_DI11, pin 14 "открыт КЭМ06.01": DD1_DI10, pin 15 "открыт КЭМ07.01": DD1_DI9, pin 16 "открыт КЭМ08.01": DD1_DI8, pin 17 "сухой ход Н02.04 (0=сух.ход)": DD5_DI.11, pin 18 "выбрать режим: Н02.04/01 - главный": N0204regimeP1M, pin 19 "выбрать режим: Н02.04/02 - главный": N0204regimeP2M, pin 20 "выбрать режим: по кол-ву включений": N0204regimeByC, pin 21 "выбрать режим: по наработке": N0204regimeWT, pin 22 "авария Н02.04/01 (0=авария)": DD5_DI.7, pin 23 "авария Н02.04/02 (0=авария)": DD5_DI.8, pin 24 "сброс аварий": alarmReset, pin 25 "сброс счетчика включений Н02.04/01": N0204resetCountP1, pin 26 "сброс счетчика включений Н02.04/02": N0204resetCountP2, pin 27 "сброс счетчика наработки Н02.04/01": N0204resetWorkTimeP1, pin 28 "сброс счетчика наработки Н02.04/02": N0204resetWorkTimeP2)
	(* Проверка, что фильтры 1 / ступени в регенерации (промывке) *)
	(* Проверка, что фильтры 2 / ступени в регенерации (промывке) *)
	(* Удержание сигнала на выключение насосов для / гарантированного сброса самоподхвата реле. *)
	(* Контроль открытия хотя бы одного из клапанов КЭМ *)
	(* сброс самоподхвата реле *)
	(* Защита от сухого хода Н02.04 / (LS02.03) 0=сух.ход *)
	#160 OR(pin 1, pin 2, pin 3, pin 4, pin 5, pin 6)
	#161 OR(#160, #162, #163)
	#162 OR(pin 7, pin 8, pin 9, pin 10, pin 11, pin 12)
	#163 OR(pin 13, pin 14, pin 15, pin 16)
	#164 N020401fTrigStop:F_TRIG(CLK: #171.pump1ON)
	#165 AND(#161, pin 17)
	#166 OR(#164.Q, #169.Q)
	#167 N0204stop:TOF(IN: #166, PT: T#1s)
	out 5 "стоп Н02.04" <= #167.Q
	#168 N0204chooseRegime:choosePumpRegime(start: #165, pump1Main: pin 18, pump2Main: pin 19, byCounter: #170, byWorkTime: pin 21)
	out 1 "выбран режим Н02.04/01 = главный" <= #168.pump1MainActive
	#169 N020402fTrigStop:F_TRIG(CLK: #171.pump2ON)
	out 2 "выбран режим Н02.04/02 = главный" <= #168.pump2MainActive
	out 3 "выбран режим по кол-ву включений" <= #168.byCounterActive
	#170 OR(pin 20, startInitializer)
	out 4 "выбран режим по наработке" <= #168.byWorkTimeActive
	#171 N0204manager:TwoPumpManager(startStopPump1: #168.startPump1, startStopPump2: #168.startPump2, alarmPump1: NOT pin 22, alarmPump2: NOT pin 23, alarmReset: pin 24, counterStart: #168.startByCounter, Pump1ResetCounter: pin 25, Pump2ResetCounter: pin 26, ValueToResetCounter: -, workTimeStart: #168.startByWorkTime, workTimePump1Reset: pin 27, workTimePump2Reset: pin 28)
	out 6 "пуск Н02.04/01" <= #171.pump1ON
	out 7 "пуск Н02.04/02" <= #171.pump2ON
	out 8 "счетчик включений Н02.04/01" <= #171.counterPump1
	out 9 "счетчик включений Н02.04/02" <= #171.counterPump2
	out 10 "счетчик наработки Н02.04/01" <= #171.currentWorkTimePump1
	out 11 "счетчик наработки Н02.04/02" <= #171.currentWorkTimePump2
END_MACRO
#172 N0204statRegimeP1M <= #159.out 1
#173 N0204statRegimeP2M <= #159.out 2
#174 N0204statRegimeByC <= #159.out 3
#175 N0204statRegimeWT <= #159.out 4
#176 DD4_DO.14 <= #159.out 5
#177 DD1_DO1 <= #159.out 6
#178 DD1_DO2 <= #159.out 7
#179 N0204counterP1 <= #159.out 8
#180 N0204counterP2 <= #159.out 9
#181 N0204workTimeP1 <= #159.out 10
#182 N0204workTimeP2 <= #159.out 11
#183 MACRO управление НД06.02 УПК(pin 1 "вход расходомера в куб/час": DD1_AI2_FT0102value, pin 2 "max производительность НД в мл/мин": ND0602setMaxDosVal, pin 3 "задание дозирования в мл/куб": ND0602setKoefProp, pin 4 "режим:1 насос главный": ND0602regimeP1M, pin 5 "режим: 2 насос главный": ND0602regimeP2M, pin 6 "режим: по наработке": ND0602regimeByWT, pin 7 "режим: по кол-ву включений": ND0602regimeByC, pin 8 "авария 1 насоса": DD6_DI.2, pin 9 "авария 2 насоса": DD6_DI.3, pin 10 "сброс аварий": alarmReset, pin 11 "сброс счетчика включений 1 насоса": ND0602resetCountP1, pin 12 "сброс ссчетчика включений 2 насоса": ND0602resetCountP2, pin 13 "сброс наработки 1 насоса": ND0602resetWorkTimeP1, pin 14 "сброс наработки 2 насоса": ND0602resetWorkTimeP2)
	(* сигнал 4...20мА на НД06.02/02 *)
	(* сигнал 4...20мА на НД06.02/01 *)
	(* Если на входе SEL = TRUE, / то нижнее значение, / иначе - то,что посередине. *)
	#184 SEL(#191.pump1ON, 0, #186.outputValue)
	#185 REAL_TO_WORD(#184)
	out 6 "выход 4...20мА насоса 1" <= #185
	#186 ND0602dosing:DosingPumpProportional(flowValue: pin 1, setMinPumpDosingValue: -, setMaxPumpDosingValue: pin 2, minOutputValue: -, maxOutputValue: -, setKoeffProportionality: pin 3, minFlowToStart: -)
	out 1 "ошибка блока дозирования" <= #186.dosingError
	#187 SEL(#191.pump2ON, 0, #186.outputValue)
	#188 REAL_TO_WORD(#187)
	out 7 "выход 4...20мА насоса 2" <= #188
	#189 ND0602regime:choosePumpRegime(start: #186.startDosingPump, pump1Main: pin 4, pump2Main: pin 5, byCounter: #190, byWorkTime: pin 6)
	out 2 "статус: 1 насос главный" <= #189.pump1MainActive
	out 3 "статус: 2 насос главный" <= #189.pump2MainActive
	out 4 "статус: по кол-ву включений" <= #189.byCounterActive
	#190 OR(pin 7, startInitializer)
	out 5 "статус: по наработке" <= #189.byWorkTimeActive
	#191 ND0602manager:TwoPumpManager(startStopPump1: #189.startPump1, startStopPump2: #189.startPump2, alarmPump1: #192, alarmPump2: #193, alarmReset: pin 10, counterStart: #189.startByCounter, Pump1ResetCounter: pin 11, Pump2ResetCounter: pin 12, ValueToResetCounter: -, workTimeStart: #189.startByWorkTime, workTimePump1Reset: pin 13, workTimePump2Reset: pin 14)
	out 12 "сигнал на включение насоса 1" <= #191.pump1ON
	#192 NOT(pin 8)
	out 13 "сигнал на включение насоса 2" <= #191.pump2ON
	out 8 "счетчик включений насоса 1" <= #191.counterPump1
	#193 NOT(pin 9)
	out 9 "счетчик включений насоса 2" <= #191.counterPump2
	out 10 "счетчик наработки насоса 1" <= #191.currentWorkTimePump1
	out 11 "счетчик наработки насоса 2" <= #191.currentWorkTimePump2
END_MACRO
#194 ND0602dosingError <= #183.out 1
#195 ND0602statRegimeP1M <= #183.out 2
#196 ND0602statRegimeP2M <= #183.out 3
#197 ND0602statRegimeByC <= #183.out 4
#198 ND0602statRegimeByWT <= #183.out 5
#199 DD10_AO1 <= #183.out 6
#200 DD10_AO2 <= #183.out 7
#201 ND0602counterP1 <= #183.out 8
#202 ND0602counterP2 <= #183.out 9
#203 ND0602workTimeP1 <= #183.out 10
#204 ND0602workTimeP2 <= #183.out 11
#205 DD4_DO.6 <= #183.out 12
#206 DD4_DO.7 <= #183.out 13
#207 OR(errorToOpenZDE0301, errorToCloseZDE0301, errorToOpenZDE0302, errorToCloseZDE0302)
#208 OR(DD5_DI.27, #207)
#209 OR(#207, DD5_DI.29)
#210 MACRO Работа УФО03.01(pin 1 "Работа УФО03.01/01": statusUFO030101started, pin 2 "Работа УФО03.01/02": statusUFO030102started, pin 3 "Значение расхода от FT01.02": DD1_AI2_FT0102value, pin 4 "мин.допустимый расход для насосов Н01.05": N0105minFlow, pin 5 "Задержка включения УФО на создание потока": UFO0301startDelayTime, pin 6 "выбор режим: УФО03.01/01 главное": UFO0301regimeP1M, pin 7 "выбор режим: УФО03.01/02 главное": UFO0301regimeP2M, pin 8 "выбор режим: по кол-ву включений": UFO0301regimeByC, pin 9 "выбор режим: по наработке": UFO0301regimeWT, pin 10 "авария УФО03.01/01": #208, pin 11 "авария УФО03.01/02": #209, pin 12 "сброс аварий": alarmReset, pin 13 "сброс счетчика включений УФО03.01/01": UFO0301resetCountP1, pin 14 "сброс счетчика включений УФО03.01/02": UFO0301resetCountP2, pin 15 "сброс счетчика наработки УФО03.01/01": UFO0301resetWorkTimeP1, pin 16 "сброс счетчика наработки УФО03.01/02": UFO0301resetWorkTimeP2)
	(* Контроль, если УФО включили вручную, / а потока при этом нет. *)
	(* Для подачи предостережения на пульте / оператора (при необходимости), а также / сигнализации лампой АВАРИЯ. *)
	(* Задержка старта УФО *)
	(* Включаем УФО, если расходомер показывает расход больше, / чем заданный как минимально допустимый для работы насосов Н01.05. *)
	#211 OR(pin 1, pin 2)
	#212 AND(#211, #213)
	out 1 "УФО вкл без потока" <= #212
	#213 NOT(#215.Q)
	#214 GE(pin 3, pin 4)
	#215 UFO0301startDelay:TON(IN: #214, PT: pin 5)
	#216 UFO0301regimeManager:choosePumpRegime(start: #215.Q, pump1Main: pin 6, pump2Main: pin 7, byCounter: #217, byWorkTime: pin 9)
	out 2 "активен режим - главное УФО 03.01/01" <= #216.pump1MainActive
	out 3 "активен режим - главное УФО 03.01/02" <= #216.pump2MainActive
	out 4 "активен режим - по кол-ву включений" <= #216.byCounterActive
	#217 OR(startInitializer, pin 8)
	out 5 "активен режим - по наработке" <= #216.byWorkTimeActive
	#218 UFO0301manager:TwoPumpManager(startStopPump1: #216.startPump1, startStopPump2: #216.startPump2, alarmPump1: pin 10, alarmPump2: pin 11, alarmReset: pin 12, counterStart: #216.startByCounter, Pump1ResetCounter: pin 13, Pump2ResetCounter: pin 14, ValueToResetCounter: -, workTimeStart: #216.startByWorkTime, workTimePump1Reset: pin 15, workTimePump2Reset: pin 16)
	out 6 "авт. пуск УФО03.01/01" <= #218.pump1ON
	out 7 "авт. пуск УФО03.01/02" <= #218.pump2ON
	out 8 "счетчик включений УФО03.01/01" <= #218.counterPump1
	out 9 "счетчик включений УФО03.01/02" <= #218.counterPump2
	out 10 "счетчик наработки УФО03.01/01" <= #218.currentWorkTimePump1
	out 11 "счетчик наработки УФО03.01/02" <= #218.currentWorkTimePump2
END_MACRO
#219 UFO0301noFlowAttention <= #210.out 1
#220 UFO0301statRegimeP1M <= #210.out 2
#221 UFO0301statRegimeP2M <= #210.out 3
#222 UFO0301statRegimeByC <= #210.out 4
#223 UFO0301statRegimeWT <= #210.out 5
#224 UFO0301counterP1 <= #210.out 8
#225 UFO0301counterP2 <= #210.out 9
#226 UFO0301workTimeP1 <= #210.out 10
#227 UFO0301workTimeP2 <= #210.out 11
#228 MACRO работа задвижек перед УФО и автом.пуск(pin 1 "сигнал на пуск УФО03.01/01": #210.out 6, pin 2 "сигнал на пуск УФО03.01/02": #210.out 7)
	(* авт.стопУФО03.01/02 *)
	(* авт.стопУФО03.01/01 *)
	(* авт.пускУФО03.01/02 *)
	(* авт.пускУФО03.01/01 *)
	(* 1 = тест задвижек ЗДЭ / 0 = возможность автом.пуска УФО *)
	(* 1 = открыть ЗДЭ03.01 / 0 = закрыть ЗДЭ03.01 *)
	(* 1 = открыть ЗДЭ03.02 / 0 = закрыть ЗДЭ03.02 *)
	#229 NOT(testZDE03)
	#230 NOT(testZDE03)
	#231 UFO030101startTrig:R_TRIG(CLK: #233)
	#232 UFO030101start <= #231.Q
	#233 AND(#229, #236, DD1_DI12)
	#234 UFO030101stopTrig:F_TRIG(CLK: #233)
	#235 UFO030101stop <= #234.Q
	#236 SEL(testZDE03, pin 1, manualZDE0301)
	#237 ZDE0301:SimpleValve(inputOpen: #236, inputClose: NOT #236, statusOpen: DD1_DI12, statusClose: DD1_DI13, reset: alarmReset, timeToOpenClose: timeToOpenCloseValve)
	#238 DD4_DO.16 <= #237.outputOpen
	#239 DD4_DO.17 <= #237.outputClose
	#240 errorToOpenZDE0301 <= #237.errorToOpen
	#241 errorToCloseZDE0301 <= #237.errorToClose
	#242 UFO030102startTrig:R_TRIG(CLK: #244)
	#243 UFO030102start <= #242.Q
	#244 AND(#230, #247, DD1_DI14)
	#245 UFO030102stopTrig:F_TRIG(CLK: #244)
	#246 UFO030102stop <= #245.Q
	#247 SEL(testZDE03, pin 2, manualZDE0302)
	#248 ZDE0302:SimpleValve(inputOpen: #247, inputClose: NOT #247, statusOpen: DD1_DI14, statusClose: DD1_DI15, reset: alarmReset, timeToOpenClose: timeToOpenCloseValve)
	#249 DD4_DO.18 <= #248.outputOpen
	#250 DD4_DO.19 <= #248.outputClose
	#251 errorToOpenZDE0302 <= #248.errorToOpen
	#252 errorToCloseZDE0302 <= #248.errorToClose
END_MACRO
#253 MACRO управление НД06.03 УПК(pin 1 "вход расходомера в куб/час": DD1_AI1_FT0101value, pin 2 "max производительность НД в мл/мин": ND0603setMaxDosVal, pin 3 "задание дозирования в мл/куб": ND0603setKoefProp, pin 4 "режим:1 насос главный": ND0603regimeP1M, pin 5 "режим: 2 насос главный": ND0603regimeP2M, pin 6 "режим: по наработке": ND0603regimeByWT, pin 7 "режим: по кол-ву включений": ND0603regimeByC, pin 8 "авария 1 насоса": DD6_DI.4, pin 9 "авария 2 насоса": DD6_DI.5, pin 10 "сброс аварий": alarmReset, pin 11 "сброс счетчика включений 1 насоса": ND0603resetCountP1, pin 12 "сброс ссчетчика включений 2 насоса": ND0603resetCountP2, pin 13 "сброс наработки 1 насоса": ND0603resetWorkTimeP1, pin 14 "сброс наработки 2 насоса": ND0603resetWorkTimeP2)
	(* сигнал 4...20мА на НД06.03/02 *)
	(* сигнал 4...20мА на НД06.03/01 *)
	(* Если на входе SEL = TRUE, / то нижнее значение, / иначе - то,что посередине. *)
	#254 SEL(#261.pump1ON, 0, #256.outputValue)
	#255 REAL_TO_WORD(#254)
	out 6 "выход 4...20мА насоса 1" <= #255
	#256 ND0603dosing:DosingPumpProportional(flowValue: pin 1, setMinPumpDosingValue: -, setMaxPumpDosingValue: pin 2, minOutputValue: -, maxOutputValue: -, setKoeffProportionality: pin 3, minFlowToStart: -)
	out 1 "ошибка блока дозирования" <= #256.dosingError
	#257 SEL(#261.pump2ON, 0, #256.outputValue)
	#258 REAL_TO_WORD(#257)
	out 7 "выход 4...20мА насоса 2" <= #258
	#259 ND0603regime:choosePumpRegime(start: #256.startDosingPump, pump1Main: pin 4, pump2Main: pin 5, byCounter: #260, byWorkTime: pin 6)
	out 2 "статус: 1 насос главный" <= #259.pump1MainActive
	out 3 "статус: 2 насос главный" <= #259.pump2MainActive
	out 4 "статус: по кол-ву включений" <= #259.byCounterActive
	#260 OR(pin 7, startInitializer)
	out 5 "статус: по наработке" <= #259.byWorkTimeActive
	#261 ND0603manager:TwoPumpManager(startStopPump1: #259.startPump1, startStopPump2: #259.startPump2, alarmPump1: #262, alarmPump2: #263, alarmReset: pin 10, counterStart: #259.startByCounter, Pump1ResetCounter: pin 11, Pump2ResetCounter: pin 12, ValueToResetCounter: -, workTimeStart: #259.startByWorkTime, workTimePump1Reset: pin 13, workTimePump2Reset: pin 14)
	out 12 "сигнал на включение насоса 1" <= #261.pump1ON
	#262 NOT(pin 8)
	out 13 "сигнал на включение насоса 2" <= #261.pump2ON
	out 8 "счетчик включений насоса 1" <= #261.counterPump1
	#263 NOT(pin 9)
	out 9 "счетчик включений насоса 2" <= #261.counterPump2
	out 10 "счетчик наработки насоса 1" <= #261.currentWorkTimePump1
	out 11 "счетчик наработки насоса 2" <= #261.currentWorkTimePump2
END_MACRO
#264 ND0603dosingError <= #253.out 1
#265 ND0603statRegimeP1M <= #253.out 2
#266 ND0603statRegimeP2M <= #253.out 3
#267 ND0603statRegimeByC <= #253.out 4
#268 ND0603statRegimeByWT <= #253.out 5
#269 DD10_AO3 <= #253.out 6
#270 DD10_AO4 <= #253.out 7
#271 ND0603counterP1 <= #253.out 8
#272 ND0603counterP2 <= #253.out 9
#273 ND0603workTimeP1 <= #253.out 10
#274 ND0603workTimeP2 <= #253.out 11
#275 DD4_DO.8 <= #253.out 12
#276 DD4_DO.9 <= #253.out 13
#277 MACRO управление Н04.04 (дренажные)(pin 1 "защита от сухого хода Н04.04": DD5_DI.18, pin 2 "автоматич.пускН04.04": DD5_DI.19, pin 3 "режим Н04.04/01 главный": N0404regimeP1M, pin 4 "режим Н04.04/02 главный": N0404regimeP2M, pin 5 "режим по кол-ву включений": N0404regimeByC, pin 6 "режим по наработке": N0404regimeWT, pin 7 "авария Н04.04/01": DD5_DI.15, pin 8 "авария Н04.04/02": DD5_DI.14, pin 9 "сброс аварий": alarmReset, pin 10 "сброс счетчика включений Н04.04/01": N0404resetCountP1, pin 11 "сброс счетчика включений Н04.04/02": N0404resetCountP2, pin 12 "сброс счетчика наработки Н04.04/01": N0404resetWorkTimeP1, pin 13 "сброс счетчика наработки Н04.04/02": N0404resetWorkTimeP2)
	(* сбрасывает самоподхват пускового реле *)
	(* Излишняя перестраховка по сухому ходу, / на уровне реле уже все отрабатывается. *)
	(* насосы имеют электрическую блокировку / от одновременного включения *)
	(* от поплавка *)
	(* сухой ход Н04.04 / 0=защита *)
	(* 0=авария *)
	#278 NOT(pin 1)
	out 1 "стоп Н04.04" <= #278
	#279 AND(pin 1, pin 2)
	#280 N0401choosePumpRegime:choosePumpRegime(start: #279, pump1Main: pin 3, pump2Main: pin 4, byCounter: #281, byWorkTime: pin 6)
	out 2 "выбран режим: Н04.04/01 главный" <= #280.pump1MainActive
	out 3 "выбран режим: Н04.04/02 главный" <= #280.pump2MainActive
	out 4 "выбран режим: по кол-ву включений" <= #280.byCounterActive
	#281 OR(startInitializer, pin 5)
	out 5 "выбран режим: по наработке" <= #280.byWorkTimeActive
	#282 N0404twoPumpManager:TwoPumpManager(startStopPump1: #280.startPump1, startStopPump2: #280.startPump2, alarmPump1: #283, alarmPump2: #284, alarmReset: pin 9, counterStart: #280.startByCounter, Pump1ResetCounter: pin 10, Pump2ResetCounter: pin 11, ValueToResetCounter: -, workTimeStart: #280.startByWorkTime, workTimePump1Reset: pin 12, workTimePump2Reset: pin 13)
	out 6 "пуск Н04.04/01" <= #282.pump1ON
	#283 NOT(pin 7)
	out 7 "пуск Н04.04/02" <= #282.pump2ON
	out 8 "счетчик кол-ва включений Н04.04/01" <= #282.counterPump1
	#284 NOT(pin 8)
	out 9 "счетчик кол-ва включений Н04.04/02" <= #282.counterPump2
	out 10 "счетчик времени наработки Н04.04/01" <= #282.currentWorkTimePump1
	out 11 "счетчик времени наработки Н04.04/02" <= #282.currentWorkTimePump2
END_MACRO
#285 DD4_DO.15 <= #277.out 1
#286 N0404statRegimeP1M <= #277.out 2
#287 N0404statRegimeP2M <= #277.out 3
#288 N0404statRegimeByC <= #277.out 4
#289 N0404statRegimeWT <= #277.out 5
#290 DD1_DO5 <= #277.out 6
#291 DD1_DO6 <= #277.out 7
#292 N0404counterP1 <= #277.out 8
#293 N0404counterP2 <= #277.out 9
#294 N0404workTimeP1 <= #277.out 10
#295 N0404workTimeP2 <= #277.out 11
#296 MACRO управление НД07.03 УПЩ (поддержка рН, ПИД-регулятор)(pin 1 "вход рН-метра QE01.01": DD1_AI3_QE0101value, pin 2 "уставка рН": ND0703pHsetValue, pin 3 "режим:1 насос главный": ND0703regimeP1M, pin 4 "режим: 2 насос главный": ND0703regimeP2M, pin 5 "режим: по наработке": ND0703regimeByWT, pin 6 "режим: по кол-ву включений": ND0703regimeByC, pin 7 "авария 1 насоса": DD6_DI.6, pin 8 "авария 2 насоса": DD6_DI.7, pin 9 "сброс аварий": alarmReset, pin 10 "сброс счетчика включений 1 насоса": ND0703resetCountP1, pin 11 "сброс счетчика включений 2 насоса": ND0703resetCountP2, pin 12 "сброс наработки 1 насоса": ND0703resetWorkTimeP1, pin 13 "сброс наработки 2 насоса": ND0703resetWorkTimeP2, pin 14 "ручное управл.выходом Y (4...20мА)": ND0703YoutManual, pin 15 "1=ручное/0=автомат.управл.": ND0703YmanAuto, pin 16 "вход расходомера FT01.01 (куб.м/час)": DD1_AI1_FT0101value, pin 17 "коэфф.I": ND0703koeffI, pin 18 "коэфф.D": ND0703koeffD, pin 19 "коэфф.Р": ND0703koeffP)
	(* сигнал 4...20мА на НД07.03/02 *)
	(* сигнал 4...20мА на НД07.03/01 *)
	(* Если на входе SEL = TRUE, / то нижнее значение, / иначе - то,что посередине. *)
	(* min расход в кубометрах в час / для неачала дозирования. *)
	#297 ND0703pidReg:PID(ACTUAL: pin 1, SET_POINT: pin 2, KP: pin 19, TN: pin 17, TV: pin 18, Y_MANUAL: pin 14, Y_OFFSET: 12, Y_MIN: 4, Y_MAX: 20, MANUAL: pin 15, RESET: #297.OVERFLOW)
	#298 SEL(#305.pump1ON, 0, #297.Y)
	#299 REAL_TO_WORD(#298)
	out 5 "выход 4...20мА насоса 1" <= #299
	#300 SEL(#305.pump2ON, 0, #297.Y)
	#301 REAL_TO_WORD(#300)
	out 6 "выход 4...20мА насоса 2" <= #301
	#302 GE(pin 16, 10)
	#303 ND0703regime:choosePumpRegime(start: #302, pump1Main: pin 3, pump2Main: pin 4, byCounter: #304, byWorkTime: pin 5)
	out 1 "статус: 1 насос главный" <= #303.pump1MainActive
	out 2 "статус: 2 насос главный" <= #303.pump2MainActive
	out 3 "статус: по кол-ву включений" <= #303.byCounterActive
	out 4 "статус: по наработке" <= #303.byWorkTimeActive
	#304 OR(pin 6, startInitializer)
	#305 ND0703manager:TwoPumpManager(startStopPump1: #303.startPump1, startStopPump2: #303.startPump2, alarmPump1: #306, alarmPump2: #307, alarmReset: pin 9, counterStart: #303.startByCounter, Pump1ResetCounter: pin 10, Pump2ResetCounter: pin 11, ValueToResetCounter: -, workTimeStart: #303.startByWorkTime, workTimePump1Reset: pin 12, workTimePump2Reset: pin 13)
	out 11 "сигнал на включение насоса 1" <= #305.pump1ON
	#306 NOT(pin 7)
	out 12 "сигнал на включение насоса 2" <= #305.pump2ON
	out 7 "счетчик включений насоса 1" <= #305.counterPump1
	#307 NOT(pin 8)
	out 8 "счетчик включений насоса 2" <= #305.counterPump2
	out 9 "счетчик наработки насоса 1" <= #305.currentWorkTimePump1
	out 10 "счетчик наработки насоса 2" <= #305.currentWorkTimePump2
END_MACRO
#308 ND0703statRegimeP1M <= #296.out 1
#309 ND0703statRegimeP2M <= #296.out 2
#310 ND0703statRegimeByC <= #296.out 3
#311 ND0703statRegimeByWT <= #296.out 4
#312 DD10_AO5 <= #296.out 5
#313 DD10_AO6 <= #296.out 6
#314 ND0703counterP1 <= #296.out 7
#315 ND0703counterP2 <= #296.out 8
#316 ND0703workTimeP1 <= #296.out 9
#317 ND0703workTimeP2 <= #296.out 10
#318 DD4_DO.10 <= #296.out 11
#319 DD4_DO.11 <= #296.out 12
#320 MACRO импульсный счетчик FQS0301(pin 1 "вход от счетчика": DD6_DI.19, pin 2 "вес импульса счетчика": FQS0301impulsValue, pin 3 "сброс счетчика": FQS0301reset, pin 4 "величина коррекции счетчика": FQS0301correction, pin 5 "прибавить коррекцию": FQS0301addCorrection, pin 6 "вычесть коррекцию": FQS0301deleteCorrection)
	(* сброс показаний счетчика *)
	(* значение в REAL (в какой-то момент начинает / отображаться в экспоненциальной форме) *)
	(* Если в результате коррекции накопленная сумма станет меньше нуля, то она принудительно станет равна нулю. *)
	(* коррекция показаний счетчика. *)
	(* число, коорое будем прибавлять или / вычитать из накопленной суммы стоков. *)
	#321 FQS0301rTrig:R_TRIG(CLK: pin 1)
	#322 ADD(EN: #321.Q, FQS0301totalAmount, pin 2)
	out 1 "накопленная сумма стоков (REAL)" <= #322
	#323 FQS0301resetRtrig:R_TRIG(CLK: pin 3)
	#324 MOVE(EN: #323.Q, 0)
	#325 FQS0301totalAmount <= #324
	#326 FQS0301addCorrRtrig:R_TRIG(CLK: pin 5)
	#327 ADD(EN: #326.Q, FQS0301totalAmount, pin 4)
	#328 FQS0301totalAmount <= #327
	#329 FQS0301deleteCorrRtrig:R_TRIG(CLK: pin 6)
	#330 SUB(EN: #329.Q, FQS0301totalAmount, pin 4)
	#331 FQS0301totalAmount <= #330
	#332 LT(FQS0301totalAmount, 0)
	#333 MOVE(EN: #332, 0)
	#334 FQS0301totalAmount <= #333
END_MACRO
#335 FQS0301totalAmount <= #320.out 1
#336 MACRO управление НД08.03 УПФ(pin 1 "вход расходомера в куб/час": DD1_AI1_FT0101value, pin 2 "max производительность НД в мл/мин": ND0803setMaxDosVal, pin 3 "задание дозирования в мл/куб": ND0803setKoefProp, pin 4 "режим:1 насос главный": ND0803regimeP1M, pin 5 "режим: 2 насос главный": ND0803regimeP2M, pin 6 "режим: по наработке": ND0803regimeByWT, pin 7 "режим: по кол-ву включений": ND0803regimeByC, pin 8 "авария 1 насоса": DD5_DI.12, pin 9 "авария 2 насоса": DD5_DI.13, pin 10 "сброс аварий": alarmReset, pin 11 "сброс счетчика включений 1 насоса": ND0803resetCountP1, pin 12 "сброс ссчетчика включений 2 насоса": ND0803resetCountP2, pin 13 "сброс наработки 1 насоса": ND0803resetWorkTimeP1, pin 14 "сброс наработки 2 насоса": ND0803resetWorkTimeP2, pin 15 "сухой ход 1 насоса": DD1_DI6, pin 16 "сухой ход 2 насоса": DD1_DI7)
	(* сигнал 4...20мА на НД08.03/02 *)
	(* сигнал 4...20мА на НД08.03/01 *)
	(* Если на входе SEL = TRUE, / то нижнее значение, / иначе - то,что посередине. *)
	#337 SEL(#346.pump1ON, 0, #338.outputValue)
	out 6 "выход 4...20мА насоса 1" <= #337
	#338 ND0803dosing:DosingPumpProportional(flowValue: pin 1, setMinPumpDosingValue: -, setMaxPumpDosingValue: pin 2, minOutputValue: -, maxOutputValue: -, setKoeffProportionality: pin 3, minFlowToStart: -)
	out 1 "ошибка блока дозирования" <= #338.dosingError
	#339 SEL(#346.pump2ON, 0, #338.outputValue)
	out 7 "выход 4...20мА насоса 2" <= #339
	#340 ND0803regime:choosePumpRegime(start: #338.startDosingPump, pump1Main: pin 4, pump2Main: pin 5, byCounter: #341, byWorkTime: pin 6)
	out 2 "статус: 1 насос главный" <= #340.pump1MainActive
	out 3 "статус: 2 насос главный" <= #340.pump2MainActive
	out 4 "статус: по кол-ву включений" <= #340.byCounterActive
	#341 OR(pin 7, startInitializer)
	out 5 "статус: по наработке" <= #340.byWorkTimeActive
	out 12 "сигнал на включение насоса 1" <= #346.pump1ON
	#342 NOT(pin 8)
	#343 OR(#342, pin 15)
	out 13 "сигнал на включение насоса 2" <= #346.pump2ON
	#344 NOT(pin 9)
	#345 OR(#344, pin 16)
	#346 ND0803manager:TwoPumpManager(startStopPump1: #340.startPump1, startStopPump2: #340.startPump2, alarmPump1: #343, alarmPump2: #345, alarmReset: pin 10, counterStart: #340.startByCounter, Pump1ResetCounter: pin 11, Pump2ResetCounter: pin 12, ValueToResetCounter: -, workTimeStart: #340.startByWorkTime, workTimePump1Reset: pin 13, workTimePump2Reset: pin 14)
	out 8 "счетчик включений насоса 1" <= #346.counterPump1
	out 9 "счетчик включений насоса 2" <= #346.counterPump2
	out 10 "счетчик наработки насоса 1" <= #346.currentWorkTimePump1
	out 11 "счетчик наработки насоса 2" <= #346.currentWorkTimePump2
END_MACRO
#347 ND0803dosingError <= #336.out 1
#348 ND0803statRegimeP1M <= #336.out 2
#349 ND0803statRegimeP2M <= #336.out 3
#350 ND0803statRegimeByC <= #336.out 4
#351 ND0803statRegimeByWT <= #336.out 5
#352 DD1_AO1 <= #336.out 6
#353 DD1_AO2 <= #336.out 7
#354 ND0803counterP1 <= #336.out 8
#355 ND0803counterP2 <= #336.out 9
#356 ND0803workTimeP1 <= #336.out 10
#357 ND0803workTimeP2 <= #336.out 11
#358 DD1_DO3 <= #336.out 12
#359 DD1_DO4 <= #336.out 13
#360 AND(DD1_DI5, DD1_DI4, DD6_DI.11)
#361 DD1_DO8 <= #360
#362 EQ(lastError, 0)
#363 alarmPLKnetworkDelay:TOF(IN: #362, PT: T#20s)
#364 NOT(#363.Q)
#365 alarmPLKnetwork <= #364
#366 MACRO управление НД08.04 УПФ(pin 1 "насос Н04.01 работает": DD7_DI.13, pin 2 "авария НД08.04": DD6_DI.16, pin 3 "уставкаНД08.04(0...100%)": ND0804doseValue)
	(* Преобразует сигнал 0...100 / пропорционально в 4...20мА *)
	#367 AND(pin 1, pin 2)
	out 1 "пуск/стоп НД08.04" <= #367
	#368 ND0804linearTransformator:LIN_TRAFO(IN: pin 3, IN_MIN: 0, IN_MAX: 100, OUT_MIN: 4, OUT_MAX: 20)
	#369 REAL_TO_WORD(#368.OUT)
	out 2 "управление НД08.04 (4...20мА)" <= #369
	out 3 "ошибка блока дозирования" <= #368.ERROR
END_MACRO
#370 DD4_DO.12 <= #366.out 1
#371 DD10_AO7 <= #366.out 2
#372 ND0804dosingError <= #366.out 3
#373 NOT(DD6_DI.0)
#374 alarmND050201 <= #373
#375 NOT(DD6_DI.23)
#376 alarmFS020102 <= #375
#377 NOT(DD9_DI.14)
#378 alarmZDE0211power <= #377
#379 NOT(DD6_DI.1)
#380 alarmND050202 <= #379
#381 NOT(DD6_DI.25)
#382 alarmFS020103 <= #381
#383 NOT(DD9_DI.15)
#384 alarmZDE0212power <= #383
#385 NOT(DD6_DI.2)
#386 alarmND060201 <= #385
#387 NOT(DD6_DI.27)
#388 alarmFS020104 <= #387
#389 NOT(DD9_DI.16)
#390 alarmZDE0213power <= #389
#391 NOT(DD6_DI.3)
#392 alarmND060202 <= #391
#393 NOT(DD6_DI.29)
#394 alarmFS020105 <= #393
#395 NOT(DD9_DI.17)
#396 alarmZDE0214power <= #395
#397 MACRO контроль включения мешалок(pin 1 "работа НД06.02/01": DD4_DO.6, pin 2 "работа НД06.02/02": DD4_DO.7, pin 3 "работа НД06.03/01": DD4_DO.8, pin 4 "работа НД06.03/02": DD4_DO.9, pin 5 "работа мешалки М06.04": DD5_DI.21, pin 6 "работа НД07.03/01": DD4_DO.10, pin 7 "работа НД07.03/02": DD4_DO.11, pin 8 "работа мешалки М07.02": DD5_DI.23, pin 9 "работа НД08.03/01": DD1_DO3, pin 10 "работа НД08.03/02": DD1_DO4, pin 11 "работа НД08.04": DD4_DO.12, pin 12 "работа мешалки М08.02": DD5_DI.25)
	#398 OR(pin 1, pin 2, pin 3, pin 4)
	#399 AND(#398, #400)
	out 1 "дозирования при выключенной М06.04" <= #399
	#400 NOT(pin 5)
	#401 OR(pin 6, pin 7)
	#402 AND(#401, #403)
	out 2 "дозирования при выключенной М07.02" <= #402
	#403 NOT(pin 8)
	#404 OR(pin 9, pin 10, pin 11)
	#405 AND(#404, #406)
	out 3 "дозирования при выключенной М08.02" <= #405
	#406 NOT(pin 12)
END_MACRO
#407 M0604attention <= #397.out 1
#408 M0702attention <= #397.out 2
#409 M0802attention <= #397.out 3
#410 NOT(DD6_DI.4)
#411 alarmND060301 <= #410
#412 NOT(DD6_DI.31)
#413 alarmFS020106 <= #412
#414 NOT(DD9_DI.18)
#415 alarmZDE0215power <= #414
#416 NOT(DD6_DI.5)
#417 alarmND060302 <= #416
#418 NOT(DD7_DI.1)
#419 alarmFS020201 <= #418
#420 NOT(DD9_DI.19)
#421 alarmZDE0216power <= #420
#422 NOT(DD6_DI.6)
#423 alarmND070301 <= #422
#424 NOT(DD7_DI.3)
#425 alarmFS020202 <= #424
#426 NOT(DD9_DI.20)
#427 alarmZDE0217power <= #426
#428 NOT(DD6_DI.7)
#429 alarmND070302 <= #428
#430 NOT(DD7_DI.5)
#431 alarmFS020203 <= #430
#432 NOT(DD9_DI.21)
#433 alarmZDE0218power <= #432
#434 NOT(DD5_DI.12)
#435 alarmND080301 <= #434
#436 NOT(DD7_DI.7)
#437 alarmFS020204 <= #436
#438 NOT(DD9_DI.22)
#439 alarmZDE0219power <= #438
#440 NOT(DD5_DI.13)
#441 alarmND080302 <= #440
#442 NOT(DD7_DI.9)
#443 alarmFS020205 <= #442
#444 NOT(DD9_DI.23)
#445 alarmZDE0220power <= #444
#446 NOT(DD6_DI.16)
#447 alarmND0804 <= #446
#448 NOT(DD7_DI.11)
#449 alarmFS020206 <= #448
#450 NOT(DD9_DI.24)
#451 alarmZDE0221power <= #450
#452 NOT(DD6_DI.11)
#453 alarmOGM0104overload <= #452
#454 NOT(DD9_DI.4)
#455 alarmZDE0201power <= #454
#456 NOT(DD9_DI.25)
#457 alarmZDE0222power <= #456
#458 MACRO переменные для обмена с панелью()
	#459 MACRO PSW регистры на передачу в панель (отображение)()
		(* PSW регистры на передачу в панель (отображение) *)
		(* panFQS0301totalAmount - переменная отображена сразу на выходе соответствующего макроса (учет очищенных стоков). / Здесь не хранится. *)
		#460 panFT0101value <= DD1_AI1_FT0101value
		#461 panQE0101value <= DD1_AI3_QE0101value
		#462 panFT0102value <= DD1_AI2_FT0102value
		#463 panQE0102value <= DD1_AI4_QE0102value
		#464 panFPKpressureValue <= DD1_AI5_FPKpressureValue
		#465 panFQS0301total <= FQS0301totalAmount
		#466 panTemperature <= temperatureValue
		#467 MACRO Время наработки и кол-во включений агрегатов()
			#468 workTimeND050201:TimeFromWorkTime(input: ND0502workTimeP1)
			#469 panND050201workDays <= #468.days
			#470 panND050201workHours <= #468.hours
			#471 panND050201workMinutes <= #468.minutes
			#472 panND050201workSeconds <= #468.seconds
			#473 workTimeND050202:TimeFromWorkTime(input: ND0502workTimeP2)
			#474 panND050202workDays <= #473.days
			#475 panND050202workHours <= #473.hours
			#476 panND050202workMinutes <= #473.minutes
			#477 panND050202workSeconds <= #473.seconds
			#478 panND0502counterP1 <= ND0502counterP1
			#479 panND0502counterP2 <= ND0502counterP2
			#480 workTimeND060201:TimeFromWorkTime(input: ND0602workTimeP1)
			#481 panND060201workDays <= #480.days
			#482 panND060201workHours <= #480.hours
			#483 panND060201workMinutes <= #480.minutes
			#484 panND060201workSeconds <= #480.seconds
			#485 workTimeND060202:TimeFromWorkTime(input: ND0602workTimeP2)
			#486 panND060202workDays <= #485.days
			#487 panND060202workHours <= #485.hours
			#488 panND060202workMinutes <= #485.minutes
			#489 panND060202workSeconds <= #485.seconds
			#490 panND0602counterP1 <= ND0602counterP1
			#491 panND0602counterP2 <= ND0602counterP2
			#492 workTimeND060301:TimeFromWorkTime(input: ND0603workTimeP1)
			#493 panND060301workDays <= #492.days
			#494 panND060301workHours <= #492.hours
			#495 panND060301workMinutes <= #492.minutes
			#496 panND060301workSeconds <= #492.seconds
			#497 workTimeND060302:TimeFromWorkTime(input: ND0603workTimeP2)
			#498 panND060302workDays <= #497.days
			#499 panND060302workHours <= #497.hours
			#500 panND060302workMinutes <= #497.minutes
			#501 panND060302workSeconds <= #497.seconds
			#502 panND0603counterP1 <= ND0603counterP1
			#503 panND0603counterP2 <= ND0603counterP2
			#504 workTimeND070301:TimeFromWorkTime(input: ND0703workTimeP1)
			#505 panND070301workDays <= #504.days
			#506 panND070301workHours <= #504.hours
			#507 panND070301workMinutes <= #504.minutes
			#508 panND070301workSeconds <= #504.seconds
			#509 workTimeND070302:TimeFromWorkTime(input: ND0703workTimeP2)
			#510 panND070302workDays <= #509.days
			#511 panND070302workHours <= #509.hours
			#512 panND070302workMinutes <= #509.minutes
			#513 panND070302workSeconds <= #509.seconds
			#514 panND0703counterP1 <= ND0703counterP1
			#515 panND0703counterP2 <= ND0703counterP2
			#516 workTimeND080301:TimeFromWorkTime(input: ND0803workTimeP1)
			#517 panND080301workDays <= #516.days
			#518 panND080301workHours <= #516.hours
			#519 panND080301workMinutes <= #516.minutes
			#520 panND080301workSeconds <= #516.seconds
			#521 workTimeND080302:TimeFromWorkTime(input: ND0803workTimeP2)
			#522 panND080302workDays <= #521.days
			#523 panND080302workHours <= #521.hours
			#524 panND080302workMinutes <= #521.minutes
			#525 panND080302workSeconds <= #521.seconds
			#526 panND0803counterP1 <= ND0803counterP1
			#527 panND0803counterP2 <= ND0803counterP2
			#528 workTimeN010501:TimeFromWorkTime(input: N0105workTimeP1)
			#529 panN010501workDays <= #528.days
			#530 panN010501workHours <= #528.hours
			#531 panN010501workMinutes <= #528.minutes
			#532 panN010501workSeconds <= #528.seconds
			#533 workTimeN010502:TimeFromWorkTime(input: N0105workTimeP2)
			#534 panN010502workDays <= #533.days
			#535 panN010502workHours <= #533.hours
			#536 panN010502workMinutes <= #533.minutes
			#537 panN010502workSeconds <= #533.seconds
			#538 panN0105counterP1 <= N0105counterP1
			#539 panN0105counterP2 <= N0105counterP2
			#540 workTimeN020401:TimeFromWorkTime(input: N0204workTimeP1)
			#541 panN020401workDays <= #540.days
			#542 panN020401workHours <= #540.hours
			#543 panN020401workMinutes <= #540.minutes
			#544 panN020401workSeconds <= #540.seconds
			#545 workTimeN020402:TimeFromWorkTime(input: N0204workTimeP2)
			#546 panN020402workDays <= #545.days
			#547 panN020402workHours <= #545.hours
			#548 panN020402workMinutes <= #545.minutes
			#549 panN020402workSeconds <= #545.seconds
			#550 panN0204counterP1 <= N0204counterP1
			#551 panN0204counterP2 <= N0204counterP2
			#552 workTimeN040401:TimeFromWorkTime(input: N0404workTimeP1)
			#553 panN040401workDays <= #552.days
			#554 panN040401workHours <= #552.hours
			#555 panN040401workMinutes <= #552.minutes
			#556 panN040401workSeconds <= #552.seconds
			#557 workTimeN040402:TimeFromWorkTime(input: N0404workTimeP2)
			#558 panN040402workDays <= #557.days
			#559 panN040402workHours <= #557.hours
			#560 panN040402workMinutes <= #557.minutes
			#561 panN040402workSeconds <= #557.seconds
			#562 panN0404counterP1 <= N0404counterP1
			#563 panN0404counterP2 <= N0404counterP2
			#564 workTimeUFO030101:TimeFromWorkTime(input: UFO0301workTimeP1)
			#565 panUFO030101workDays <= #564.days
			#566 panUFO030101workHours <= #564.hours
			#567 panUFO030101workMinutes <= #564.minutes
			#568 panUFO030101workSeconds <= #564.seconds
			#569 workTimeUFO030102:TimeFromWorkTime(input: UFO0301workTimeP2)
			#570 panUFO030102workDays <= #569.days
			#571 panUFO030102workHours <= #569.hours
			#572 panUFO030102workMinutes <= #569.minutes
			#573 panUFO030102workSeconds <= #569.seconds
			#574 panUFO0301counterP1 <= UFO0301counterP1
			#575 panUFO0301counterP2 <= UFO0301counterP2
		END_MACRO
		#576 panVolumeToRegen <= volumeToRegen
	END_MACRO
	#577 MACRO PSB регистры на передачу в панель (отображение)()
		(* PSB регистры на передачу в панель (отображение) *)
		#578 MACRO 8 bit output module 1()
			#579 panStartND050201 <= DD4_DO.4
			#580 panStartND050202 <= DD4_DO.5
			#581 panStartND060201 <= DD4_DO.6
			#582 panStartND060202 <= DD4_DO.7
			#583 panStartND060301 <= DD4_DO.8
			#584 panStartND060302 <= DD4_DO.9
			#585 panStartM0604 <= DD5_DI.21
			#586 panStartND070301 <= DD4_DO.10
		END_MACRO
		#587 MACRO 8 bit output module 2()
			#588 panStartND070302 <= DD4_DO.11
			#589 panStartM0702 <= DD5_DI.23
			#590 panStartND080301 <= DD1_DO3
			#591 panStartND080302 <= DD1_DO4
			#592 panStartND0804 <= DD4_DO.12
			#593 panStartM0802 <= DD5_DI.25
			#594 panStartN020401 <= DD5_DI.9
			#595 panStartN020402 <= DD5_DI.10
		END_MACRO
		#596 MACRO 8 bit output module 3()
			#597 panStartN010501 <= N0105statStartedP1
			#598 panStartN010502 <= N0105statStartedP2
			#599 panCleanFS020101 <= DD6_DI.20
			#600 panCleanFS020102 <= DD6_DI.22
			#601 panCleanFS020103 <= DD6_DI.24
			#602 panCleanFS020104 <= DD6_DI.26
			#603 panCleanFS020105 <= DD6_DI.28
			#604 panCleanFS020106 <= DD6_DI.30
		END_MACRO
		#605 MACRO 8 bit output module 4()
			#606 panCleanFS020201 <= DD7_DI. 0
			#607 panCleanFS020202 <= DD7_DI. 2
			#608 panCleanFS020203 <= DD7_DI. 4
			#609 panCleanFS020204 <= DD7_DI. 6
			#610 panCleanFS020205 <= DD7_DI. 8
			#611 panCleanFS020206 <= DD7_DI. 10
			#612 panSludgeReady <= DD7_DI.15
			#613 panStartN0401 <= DD7_DI.13
		END_MACRO
		#614 MACRO 8 bit output module 5()
			#615 panKSHE0401open <= DD9_DI.2
			#616 panFPKready <= DD7_DI.12
			#617 panFPKneedToClean <= FPKneedToClean
			#618 panStartN040401 <= DD5_DI.16
			#619 panStartN040402 <= DD5_DI.17
			#620 panStartUFO030101 <= statusUFO030101started
			#621 panStartUFO030102 <= statusUFO030102started
			#622 panAlarm <= alarm
		END_MACRO
		#623 MACRO 8 bit output module 6()
			#624 panErrorTempSensor <= DD1_AI0_error
			#625 panErrorFT0101 <= DD1_AI1_error
			#626 panErrorFT0102 <= DD1_AI2_error
			#627 panErrorQE0102 <= DD1_AI3_error
			#628 panErrorQE0102 <= DD1_AI4_error
			#629 panAlarmHighTemp <= alarmHighTemperature
			#630 panAlarmLowTemp <= alarmLowTemperature
			#631 panND0502dosingError <= ND0502dosingError
		END_MACRO
		#632 MACRO 8 bit output module 7()
			#633 panND0602dosingError <= ND0602dosingError
			#634 panND0603dosingError <= ND0603dosingError
			#635 panND0803dosingError <= ND0803dosingError
			#636 panND0804dosingError <= ND0804dosingError
			#637 panND080301emptyAlarm <= DD1_DI6
			#638 panND080302emptyAlarm <= DD1_DI7
			#639 panN010501alarm <= N010501alarm
			#640 panN010502alarm <= N010502alarm
		END_MACRO
		#641 MACRO 8 bit output module 8()
			#642 panZDE0225errorToOpen <= ZDE0225errorToOpen
			#643 panZDE0225errorToClose <= ZDE0225errorToClose
			#644 panFPKalarm <= DD7_DI.14
			#645 panFPKnotStarted <= FPKnotStarted
			#646 panErrorFPKsensor <= DD1_AI5_error
			#647 panFPKkshe0401errorToOpen <= FPKkshe0401errorToOpen
			#648 panFPKkshe0401errorToClose <= FPKkshe0401errorToClose
			#649 panUFO030101alarm <= statusUFO030101alarm
		END_MACRO
		#650 MACRO 8 bit output module 9()
			#651 panUFO030102alarm <= statusUFO030102alarm
			#652 panFilterFailToRegen020101 <= filterFailToRegen020101
			#653 panErrorToOpenZD0201 <= errorToOpenZD0201
			#654 panErrorToCloseZD0201 <= errorToCloseZD0201
			#655 panErrorToOpenZD0207 <= errorToOpenZD0207
			#656 panErrorToCloseZD0207 <= errorToCloseZD0207
			#657 panFilterFailToRegen020102 <= filterFailToRegen020102
			#658 panErrorToOpenZD0202 <= errorToOpenZD0202
		END_MACRO
		#659 MACRO 8 bit output module 10()
			#660 panErrorToCloseZD0202 <= errorToCloseZD0202
			#661 panErrorToOpenZD0208 <= errorToOpenZD0208
			#662 panErrorToCloseZD0208 <= errorToCloseZD0208
			#663 panFilterFailToRegen020103 <= filterFailToRegen020103
			#664 panErrorToOpenZD0203 <= errorToOpenZD0203
			#665 panErrorToCloseZD0203 <= errorToCloseZD0203
			#666 panErrorToOpenZD0209 <= errorToOpenZD0209
			#667 panErrorToCloseZD0209 <= errorToCloseZD0209
		END_MACRO
		#668 MACRO 8 bit output module 11()
			#669 panFilterFailToRegen020104 <= filterFailToRegen020104
			#670 panErrorToOpenZD0204 <= errorToOpenZD0204
			#671 panErrorToCloseZD0204 <= errorToCloseZD0204
			#672 panErrorToOpenZD0210 <= errorToOpenZD0210
			#673 panErrorToCloseZD0210 <= errorToCloseZD0210
			#674 panFilterFailToRegen020105 <= filterFailToRegen020105
			#675 panErrorToOpenZD0205 <= errorToOpenZD0205
			#676 panErrorToCloseZD0205 <= errorToCloseZD0205
		END_MACRO
		#677 MACRO 8 bit output module 12()
			#678 panErrorToOpenZD0211 <= errorToOpenZD0211
			#679 panErrorToCloseZD0211 <= errorToCloseZD0211
			#680 panFilterFailToRegen020106 <= filterFailToRegen020106
			#681 panErrorToOpenZD0206 <= errorToOpenZD0206
			#682 panErrorToCloseZD0206 <= errorToCloseZD0206
			#683 panErrorToOpenZD0212 <= errorToOpenZD0212
			#684 panErrorToCloseZD0212 <= errorToCloseZD0212
			#685 panFilterFailToRegen020201 <= filterFailToRegen020201
		END_MACRO
		#686 MACRO 8 bit output module 13()
			#687 panErrorToOpenZD0213 <= errorToOpenZD0213
			#688 panErrorToCloseZD0213 <= errorToCloseZD0213
			#689 panErrorToOpenZD0219 <= errorToOpenZD0219
			#690 panErrorToCloseZD0219 <= errorToCloseZD0219
			#691 panFilterFailToRegen020202 <= filterFailToRegen020202
			#692 panErrorToOpenZD0214 <= errorToOpenZD0214
			#693 panErrorToCloseZD0214 <= errorToCloseZD0214
			#694 panErrorToOpenZD0220 <= errorToOpenZD0220
		END_MACRO
		#695 MACRO 8 bit output module 14()
			#696 panErrorToCloseZD0220 <= errorToCloseZD0220
			#697 panFilterFailToRegen020203 <= filterFailToRegen020203
			#698 panErrorToOpenZD0215 <= errorToOpenZD0215
			#699 panErrorToCloseZD0215 <= errorToCloseZD0215
			#700 panErrorToOpenZD0221 <= errorToOpenZD0221
			#701 panErrorToCloseZD0221 <= errorToCloseZD0221
			#702 panFilterFailToRegen020204 <= filterFailToRegen020204
			#703 panErrorToOpenZD0216 <= errorToOpenZD0216
		END_MACRO
		#704 MACRO 8 bit output module 15()
			#705 panErrorToCloseZD0216 <= errorToCloseZD0216
			#706 panErrorToOpenZD0222 <= errorToOpenZD0222
			#707 panErrorToCloseZD0222 <= errorToCloseZD0222
			#708 panFilterFailToRegen020205 <= filterFailToRegen020205
			#709 panErrorToOpenZD0217 <= errorToOpenZD0217
			#710 panErrorToCloseZD0217 <= errorToCloseZD0217
			#711 panErrorToOpenZD0223 <= errorToOpenZD0223
			#712 panErrorToCloseZD0223 <= errorToCloseZD0223
		END_MACRO
		#713 MACRO 8 bit output module 16()
			#714 panFilterFailToRegen020206 <= filterFailToRegen020206
			#715 panErrorToOpenZD0218 <= errorToOpenZD0218
			#716 panErrorToCloseZD0218 <= errorToCloseZD0218
			#717 panErrorToOpenZD0224 <= errorToOpenZD0224
			#718 panErrorToCloseZD0224 <= errorToCloseZD0224
			#719 panAlarmPLKnetwork <= alarmPLKnetwork
			#720 panAlarmND050201 <= alarmND050201
			#721 panAlarmND050202 <= alarmND050202
		END_MACRO
		#722 MACRO 8 bit output module 17()
			#723 panAlarmND060201 <= alarmND060201
			#724 panAlarmND060202 <= alarmND060202
			#725 panAlarmND060301 <= alarmND060301
			#726 panAlarmND060302 <= alarmND060302
			#727 panAlarmND070301 <= alarmND070301
			#728 panAlarmND070302 <= alarmND070302
			#729 panAlarmND080301 <= alarmND080301
			#730 panAlarmND080302 <= alarmND080302
		END_MACRO
		#731 MACRO 8 bit output module 18()
			#732 panAlarmND0804 <= alarmND0804
			#733 panAlarmOGM0104overload <= alarmOGM0104overload
			#734 panAlarmRCHV0203overload <= alarmRCHV0203overload
			#735 panAlarmN040402 <= alarmN040402
			#736 panAlarmN040401 <= alarmN040401
			#737 panAlarmM0604 <= alarmM0604
			#738 panAlarmM0702 <= alarmM0702
			#739 panAlarmM0802 <= alarmM0802
		END_MACRO
		#740 MACRO 8 bit output module 19()
			#741 panAlarmN020401 <= alarmN020401
			#742 panAlarmN020402 <= alarmN020402
			#743 panAlarmFS020101 <= alarmFS020101
			#744 panAlarmFS020102 <= alarmFS020102
			#745 panAlarmFS020103 <= alarmFS020103
			#746 panAlarmFS020104 <= alarmFS020104
			#747 panAlarmFS020105 <= alarmFS020105
			#748 panAlarmFS020106 <= alarmFS020106
		END_MACRO
		#749 MACRO 8 bit output module 20()
			#750 panAlarmFS020201 <= alarmFS020201
			#751 panAlarmFS020202 <= alarmFS020202
			#752 panAlarmFS020203 <= alarmFS020203
			#753 panAlarmFS020204 <= alarmFS020204
			#754 panAlarmFS020205 <= alarmFS020205
			#755 panAlarmFS020206 <= alarmFS020206
			#756 panAlarmZDE0201power <= alarmZDE0201power
			#757 panAlarmZDE0202power <= alarmZDE0202power
		END_MACRO
		#758 MACRO 8 bit output module 21()
			#759 panAlarmZDE0203power <= alarmZDE0203power
			#760 panAlarmZDE0204power <= alarmZDE0204power
			#761 panAlarmZDE0205power <= alarmZDE0205power
			#762 panAlarmZDE0206power <= alarmZDE0206power
			#763 panAlarmZDE0207power <= alarmZDE0207power
			#764 panAlarmZDE0208power <= alarmZDE0208power
			#765 panAlarmZDE0209power <= alarmZDE0209power
			#766 panAlarmZDE0210power <= alarmZDE0210power
		END_MACRO
		#767 MACRO 8 bit output module 22()
			#768 panAlarmZDE0211power <= alarmZDE0211power
			#769 panAlarmZDE0212power <= alarmZDE0212power
			#770 panAlarmZDE0213power <= alarmZDE0213power
			#771 panAlarmZDE0214power <= alarmZDE0214power
			#772 panAlarmZDE0215power <= alarmZDE0215power
			#773 panAlarmZDE0216power <= alarmZDE0216power
			#774 panAlarmZDE0217power <= alarmZDE0217power
			#775 panAlarmZDE0218power <= alarmZDE0218power
		END_MACRO
		#776 MACRO 8 bit output module 23()
			#777 panAlarmZDE0219power <= alarmZDE0219power
			#778 panAlarmZDE0220power <= alarmZDE0220power
			#779 panAlarmZDE0221power <= alarmZDE0221power
			#780 panAlarmZDE0222power <= alarmZDE0222power
			#781 panAlarmZDE0223power <= alarmZDE0223power
			#782 panAlarmZDE0224power <= alarmZDE0224power
			#783 panAlarmZDE0225power <= alarmZDE0225power
			#784 panAlarmKSHE0401power <= alarmKSHE0401power
		END_MACRO
		#785 MACRO 8 bit output module 24()
			#786 panAlarmKNS <= alarmKNS
			#787 panAlarmPowerSocketFS <= alarmPowerSocketFS
			#788 panAlarmKEMvalvesPower <= alarmKEMvalvesPower
			#789 panAlarmEmergencyPressed <= alarmEmergencyPressed
			#790 panAlarmRKF <= alarmRKF
			#791 panUFO0301noFlowAttention <= UFO0301noFlowAttention
			#792 panM0604attention <= M0604attention
			#793 panM0702attention <= M0702attention
		END_MACRO
		#794 MACRO 8 bit output module 25()
			#795 panM0802attention <= M0802attention
			#796 panStatusKNS <= DD6_DI.8
			#797 panND0502statRegimeP1M <= ND0502statRegimeP1M
			#798 panND0502statRegimeP2M <= ND0502statRegimeP2M
			#799 panND0502statRegimeByC <= ND0502statRegimeByC
			#800 panND0502statRegimeByWT <= ND0502statRegimeByWT
			#801 panND0602statRegimeP1M <= ND0602statRegimeP1M
			#802 panND0602statRegimeP2M <= ND0602statRegimeP2M
		END_MACRO
		#803 MACRO 8 bit output module 26()
			#804 panND0602statRegimeByC <= ND0602statRegimeByC
			#805 panND0602statRegimeByWT <= ND0602statRegimeByWT
			#806 panND0603statRegimeP1M <= ND0603statRegimeP1M
			#807 panND0603statRegimeP2M <= ND0603statRegimeP2M
			#808 panND0603statRegimeByC <= ND0603statRegimeByC
			#809 panND0603statRegimeByWT <= ND0603statRegimeByWT
			#810 panND0703statRegimeP1M <= ND0703statRegimeP1M
			#811 panND0703statRegimeP2M <= ND0703statRegimeP2M
		END_MACRO
		#812 MACRO 8 bit output module 27()
			#813 panND0703statRegimeByC <= ND0703statRegimeByC
			#814 panND0703statRegimeByWT <= ND0703statRegimeByWT
			#815 panND0803statRegimeP1M <= ND0803statRegimeP1M
			#816 panND0803statRegimeP2M <= ND0803statRegimeP2M
			#817 panND0803statRegimeByC <= ND0803statRegimeByC
			#818 panND0803statRegimeByWT <= ND0803statRegimeByWT
			#819 panN0105statRegimeP1M <= N0105statRegimeP1M
			#820 panN0105statRegimeP2M <= N0105statRegimeP2M
		END_MACRO
		#821 MACRO 8 bit output module 28()
			#822 panN0105statRegimeByC <= N0105statRegimeByC
			#823 panN0105statRegimeByWT <= N0105statRegimeByWT
			#824 panN0204statRegimeP1M <= N0204statRegimeP1M
			#825 panN0204statRegimeP2M <= N0204statRegimeP2M
			#826 panN0204statRegimeByC <= N0204statRegimeByC
			#827 panN0204statRegimeWT <= N0204statRegimeWT
			#828 panN0404statRegimeP1M <= N0404statRegimeP1M
			#829 panN0404statRegimeP2M <= N0404statRegimeP2M
		END_MACRO
		#830 MACRO 8 bit output module 29()
			#831 panN0404statRegimeByC <= N0404statRegimeByC
			#832 panN0404statRegimeWT <= N0404statRegimeWT
			#833 panUFO0301statRegimeP1M <= UFO0301statRegimeP1M
			#834 panUFO0301statRegimeP2M <= UFO0301statRegimeP2M
			#835 panUFO0301statRegimeByC <= UFO0301statRegimeByC
			#836 panUFO0301statRegimeWT <= UFO0301statRegimeWT
			#837 panZDE0225open <= DD9_DI.0
			#838 panZDE0201open <= DD7_DI.16
		END_MACRO
		#839 MACRO 8 bit output module 30()
			#840 panZDE0201close <= DD7_DI.17
			#841 panZDE0202open <= DD7_DI.18
			#842 panZDE0202close <= DD7_DI.19
			#843 panZDE0203open <= DD7_DI.20
			#844 panZDE0203close <= DD7_DI.21
			#845 panZDE0204open <= DD7_DI.22
			#846 panZDE0204close <= DD7_DI.23
			#847 panZDE0205open <= DD7_DI.24
		END_MACRO
		#848 MACRO 8 bit output module 31()
			#849 panZDE0205close <= DD7_DI.25
			#850 panZDE0206open <= DD7_DI.26
			#851 panZDE0206close <= DD7_DI.27
			#852 panZDE0207open <= DD7_DI.28
			#853 panZDE0207close <= DD7_DI.29
			#854 panZDE0208open <= DD7_DI.30
			#855 panZDE0208close <= DD7_DI.31
			#856 panZDE0209open <= DD8_DI.0
		END_MACRO
		#857 MACRO 8 bit output module 32()
			#858 panZDE0209close <= DD8_DI.1
			#859 panZDE0210open <= DD8_DI.2
			#860 panZDE0210close <= DD8_DI.3
			#861 panZDE0211open <= DD8_DI.4
			#862 panZDE0211close <= DD8_DI.5
			#863 panZDE0212open <= DD8_DI.6
			#864 panZDE0212close <= DD8_DI.7
			#865 panZDE0213open <= DD8_DI.8
		END_MACRO
		#866 MACRO 8 bit output module 33()
			#867 panZDE0213close <= DD8_DI.9
			#868 panZDE0214open <= DD8_DI.10
			#869 panZDE0214close <= DD8_DI.11
			#870 panZDE0215open <= DD8_DI.12
			#871 panZDE0215close <= DD8_DI.13
			#872 panZDE0216open <= DD8_DI.14
			#873 panZDE0216close <= DD8_DI.15
			#874 panZDE0217open <= DD8_DI.16
		END_MACRO
		#875 MACRO 8 bit output module 34()
			#876 panZDE0217close <= DD8_DI.17
			#877 panZDE0218open <= DD8_DI.18
			#878 panZDE0218close <= DD8_DI.19
			#879 panZDE0219open <= DD8_DI.20
			#880 panZDE0219close <= DD8_DI.21
			#881 panZDE0220open <= DD8_DI.22
			#882 panZDE0220close <= DD8_DI.23
			#883 panZDE0221open <= DD8_DI.24
		END_MACRO
		#884 MACRO 8 bit output module 35()
			#885 panZDE0221close <= DD8_DI.25
			#886 panZDE0222open <= DD8_DI.26
			#887 panZDE0222close <= DD8_DI.27
			#888 panZDE0223open <= DD8_DI.28
			#889 panZDE0223close <= DD8_DI.29
			#890 panZDE0224open <= DD8_DI.30
			#891 panZDE0224close <= DD8_DI.31
			#892 panZDE0225close <= DD9_DI.1
		END_MACRO
		#893 MACRO 8 bit output module 36x()
			#894 panKSHE0401close <= DD9_DI.3
			#895 panZDE0301open <= DD1_DI12
			#896 panZDE0301close <= DD1_DI13
			#897 panZDE0302open <= DD1_DI14
			#898 panZDE0302close <= DD1_DI15
			#899 panErrorToOpenZDE0301 <= errorToOpenZDE0301
			#900 panErrorToCloseZDE0301 <= errorToCloseZDE0301
			#901 panErrorToOpenZDE0302 <= errorToOpenZDE0302
		END_MACRO
		#902 panErrorToCloseZDE0302 <= errorToCloseZDE0302
		#903 panAlarmZDE0301power <= alarmZDE0301power
		#904 panAlarmZDE0302power <= alarmZDE0302power
		#905 panUFO030101danger <= statusUFO030101danger
		#906 panUFO030102danger <= statusUFO030102danger
		#907 panUFO030101distantMode <= statusUFO030101distantMode
		#908 panUFO030102distantMode <= statusUFO030102distantMode
	END_MACRO
	#909 MACRO PFW регистры на чтение из панели (управление ПЛК)()
		#910 MUL(panTimeToOpenCloseValve, 1000)
		#911 REAL_TO_TIME(#910)
		#912 TimeToOpenCloseValve <= #911
		#913 maxTemperature <= panMaxTemperature
		#914 minTemperature <= panMinTemperature
		#915 ND0502setMaxDosVal <= panND0502setMaxDosVal
		#916 ND0502setKoefProp <= panND0502setKoefProp
		#917 ND0602setMaxDosVal <= panND0602setMaxDosVal
		#918 ND0602setKoefProp <= panND0602setKoefProp
		#919 ND0603setMaxDosVal <= panND0603setMaxDosVal
		#920 ND0603setKoefProp <= panND0603setKoefProp
		#921 ND0703pHsetValue <= panND0703pHsetValue
		#922 ND0703YoutManual <= panND0703YoutManual
		#923 ND0703koeffI <= panND0703koeffI
		#924 ND0703koeffD <= panND0703koeffD
		#925 ND0703koeffP <= panND0703koeffP
		#926 ND0803setMaxDosVal <= panND0803setMaxDosVal
		#927 ND0803setKoefProp <= panND0803setKoefProp
		#928 ND0804doseValue <= panND0804doseValue
		#929 N0105flowSetValue <= panN0105flowSetValue
		#930 N0105YoutManual <= panN0105YoutManual
		#931 N0105koeffI <= panN0105koeffI
		#932 N0105koeffD <= panN0105koeffD
		#933 N0105koeffP <= panN0105koeffP
		#934 FQS0301impulsValue <= panFQS0301impulsValue
		#935 FQS0301correction <= panFQS0301correction
		#936 MUL(panFPKtimeToWork, 1000)
		#937 REAL_TO_TIME(#936)
		#938 FPKtimeToWork <= #937
		#939 MUL(panFPKnotStartedTime, 1000)
		#940 REAL_TO_TIME(#939)
		#941 FPKnotStartedTime <= #940
		#942 FPKmaxPressureValue <= panFPKmaxPressureValue
		#943 filterValueToRegen <= panFilterValueToRegen
	END_MACRO
	#944 MACRO PSB регистры на чтение из панели (управление ПЛК)()
		(* PSB регистры на чтение из панели (управление ПЛК) *)
		#945 MACRO 8 bit input module 1()
			#1275 alarmReset <= panAlarmResetButton
			#1276 ND0502resetCountP1 <= panND0502resetCountP1
			#1277 ND0502resetCountP2 <= panND0502resetCountP2
			#1278 ND0502resetWorkTimeP1 <= panND0502resetWorkTimeP1
			#1279 ND0502resetWorkTimeP2 <= panND0502resetWorkTimeP2
			#1280 ND0502regimeP1M <= panND0502regimeP1M
			#1281 ND0502regimeP2M <= panND0502regimeP2M
			#1282 ND0502regimeByC <= panND0502regimeByC
		END_MACRO
		#946 MACRO 8 bit input module 2()
			#1283 ND0502regimeByWT <= panND0502regimeByWT
			#1284 ND0602resetCountP1 <= panND0602resetCountP1
			#1285 ND0602resetCountP2 <= panND0602resetCountP2
			#1286 ND0602resetWorkTimeP1 <= panND0602resetWorkTimeP1
			#1287 ND0602resetWorkTimeP2 <= panND0602resetWorkTimeP2
			#1288 ND0602regimeP1M <= panND0602regimeP1M
			#1289 ND0602regimeP2M <= panND0602regimeP2M
			#1290 ND0602regimeByC <= panND0602regimeByC
		END_MACRO
		#947 MACRO 8 bit input module 3()
			#1291 ND0602regimeByWT <= panND0602regimeByWT
			#1292 ND0603resetCountP1 <= panND0603resetCountP1
			#1293 ND0603resetCountP2 <= panND0603resetCountP2
			#1294 ND0603resetWorkTimeP1 <= panND0603resetWorkTimeP1
			#1295 ND0603resetWorkTimeP2 <= panND0603resetWorkTimeP2
			#1296 ND0603regimeP1M <= panND0603regimeP1M
			#1297 ND0603regimeP2M <= panND0603regimeP2M
			#1298 ND0603regimeByC <= panND0603regimeByC
		END_MACRO
		#948 MACRO 8 bit input module 4()
			#1299 ND0603regimeByWT <= panND0603regimeByWT
			#1300 ND0703resetCountP1 <= panND0703resetCountP1
			#1301 ND0703resetCountP2 <= panND0703resetCountP2
			#1302 ND0703resetWorkTimeP1 <= panND0703resetWorkTimeP1
			#1303 ND0703resetWorkTimeP2 <= panND0703resetWorkTimeP2
			#1304 ND0703regimeP1M <= panND0703regimeP1M
			#1305 ND0703regimeP2M <= panND0703regimeP2M
			#1306 ND0703regimeByC <= panND0703regimeByC
		END_MACRO
		#949 MACRO 8 bit input module 5()
			#1307 ND0703regimeByWT <= panND0703regimeByWT
			#1308 ND0703YmanAuto <= panND0703YmanAuto
			#1309 ND0803resetCountP1 <= panND0803resetCountP1
			#1310 ND0803resetCountP2 <= panND0803resetCountP2
			#1311 ND0803resetWorkTimeP1 <= panND0803resetWorkTimeP1
			#1312 ND0803resetWorkTimeP2 <= panND0803resetWorkTimeP2
			#1313 ND0803regimeP1M <= panND0803regimeP1M
			#1314 ND0803regimeP2M <= panND0803regimeP2M
		END_MACRO
		#950 MACRO 8 bit input module 6()
			#1315 ND0803regimeByC <= panND0803regimeByC
			#1316 ND0803regimeByWT <= panND0803regimeByWT
			#1317 N0105resetCountP1 <= panN0105resetCountP1
			#1318 N0105resetCountP2 <= panN0105resetCountP2
			#1319 N0105resetWorkTimeP1 <= panN0105resetWorkTimeP1
			#1320 N0105resetWorkTimeP2 <= panN0105resetWorkTimeP2
			#1321 N0105regimeByC <= panN0105regimeByC
			#1322 N0105regimeByWT <= panN0105regimeByWT
		END_MACRO
		#951 MACRO 8 bit input module 7()
			#1323 N0105YmanAuto <= panN0105YmanAuto
			#1324 N0204resetCountP1 <= panN0204resetCountP1
			#1325 N0204resetCountP2 <= panN0204resetCountP2
			#1326 N0204resetWorkTimeP1 <= panN0204resetWorkTimeP1
			#1327 N0204resetWorkTimeP2 <= panN0204resetWorkTimeP2
			#1328 N0204regimeP1M <= panN0204regimeP1M
			#1329 N0204regimeP2M <= panN0204regimeP2M
			#1330 N0204regimeByC <= panN0204regimeByC
		END_MACRO
		#952 MACRO 8 bit input module 8()
			#1331 N0204regimeWT <= panN0204regimeWT
			#1332 UFO0301resetCountP1 <= panUFO0301resetCountP1
			#1333 UFO0301resetCountP2 <= panUFO0301resetCountP2
			#1334 UFO0301resetWorkTimeP1 <= panUFO0301resetWorkTimeP1
			#1335 UFO0301resetWorkTimeP2 <= panUFO0301resetWorkTimeP2
			#1336 UFO0301regimeP1M <= panUFO0301regimeP1M
			#1337 UFO0301regimeP2M <= panUFO0301regimeP2M
			#1338 UFO0301regimeByC <= panUFO0301regimeByC
		END_MACRO
		#953 MACRO 8 bit input module 9()
			#1339 UFO0301regimeWT <= panUFO0301regimeWT
			#1340 N0404resetCountP1 <= panN0404resetCountP1
			#1341 N0404resetCountP2 <= panN0404resetCountP2
			#1342 N0404resetWorkTimeP1 <= panN0404resetWorkTimeP1
			#1343 N0404resetWorkTimeP2 <= panN0404resetWorkTimeP2
			#1344 N0404regimeP1M <= panN0404regimeP1M
			#1345 N0404regimeP2M <= panN0404regimeP2M
			#1346 N0404regimeByC <= panN0404regimeByC
		END_MACRO
		#954 MACRO 8 bit input module 10-11()
			(* одули 10 и 11 заполнены переменными для тестирования задвижек. / Здесь они не показаны, т.к. спешка. / Они вставлены напрямую в макросы управления промывкой фильтров. / testValvesFS020101 - testValvesFS020206 (PSB612-623) *)
			#1347 N0404regimeWT <= panN0404regimeWT
			#1348 FQS0301reset <= panFQS0301reset
			#1349 FQS0301addCorrection <= panFQS0301addCorrection
			#1350 FQS0301deleteCorrection <= panFQS0301deleteCorrection
		END_MACRO
		#955 testKSHE0401 <= panTestKSHE0401
		#956 testZDE0225 <= panTestZDE0225
		#957 testZDE03 <= panTestZDE03
		#958 manualZDE0301 <= panManualZDE0301
		#959 manualZDE0302 <= panManualZDE0302
	END_MACRO
END_MACRO
#960 NOT(DD6_DI.13)
#961 alarmRCHV0203overload <= #960
#962 NOT(DD9_DI.5)
#963 alarmZDE0202power <= #962
#964 NOT(DD9_DI.26)
#965 alarmZDE0223power <= #964
#966 MACRO переменные на диспетчеризацию()
	#967 remFT0101value <= DD1_AI1_FT0101value
	#968 remFQS0301totalAmount <= FQS0301totalAmount
	#969 remTemperatureValue <= temperatureValue
	#970 remStatusN010501started <= N0105statStartedP1
	#971 remStatusN010502started <= N0105statStartedP2
	#972 remStatusUFO030101started <= statusUFO030101started
	#973 remStatusUFO030102started <= statusUFO030102started
	#974 remAlarm <= Alarm
	#975 remN010501alarm <= N010501alarm
	#976 remN010502alarm <= N010502alarm
	#977 remFPKalarm <= DD7_DI.14
	#978 remUFO030101alarm <= statusUFO030101alarm
	#979 remUFO030102alarm <= statusUFO030102alarm
	#980 remAlarmEmergencyPressed <= alarmEmergencyPressed
	#981 remAlarmOOGM0104overload <= DD6_DI.11
	#982 remAlarmRCHV0203overload <= DD6_DI.13
END_MACRO
#983 NOT(DD5_DI.14)
#984 alarmN040402 <= #983
#985 NOT(DD9_DI.6)
#986 alarmZDE0203power <= #985
#987 NOT(DD9_DI.27)
#988 alarmZDE0224power <= #987
#989 NOT(DD5_DI.15)
#990 alarmN040401 <= #989
#991 NOT(DD9_DI.7)
#992 alarmZDE0204power <= #991
#993 NOT(DD9_DI.28)
#994 alarmZDE0225power <= #993
#995 NOT(DD5_DI.20)
#996 alarmM0604 <= #995
#997 NOT(DD9_DI.8)
#998 alarmZDE0205power <= #997
#999 NOT(DD9_DI.29)
#1000 alarmKSHE0401power <= #999
#1001 NOT(DD5_DI.22)
#1002 alarmM0702 <= #1001
#1003 NOT(DD9_DI.9)
#1004 alarmZDE0206power <= #1003
#1005 NOT(DD6_DI.9)
#1006 alarmKNS <= #1005
#1007 NOT(DD5_DI.24)
#1008 alarmM0802 <= #1007
#1009 NOT(DD9_DI.10)
#1010 alarmZDE0207power <= #1009
#1011 NOT(DD6_DI.17)
#1012 alarmPowerSocketFS <= #1011
#1013 NOT(DD5_DI.7)
#1014 alarmN020401 <= #1013
#1015 NOT(DD9_DI.11)
#1016 alarmZDE0208power <= #1015
#1017 NOT(DD6_DI.18)
#1018 alarmKEMvalvesPower <= #1017
#1019 NOT(DD5_DI.8)
#1020 alarmN020402 <= #1019
#1021 NOT(DD9_DI.12)
#1022 alarmZDE0209power <= #1021
#1023 NOT(DD1_DI4)
#1024 alarmEmergencyPressed <= #1023
#1025 GT(DD1_AI2_FT0102value, 0)
#1026 filterPulserGen:PulsePerSec(start: #1025)
#1027 DIV(DD1_AI2_FT0102value, 3600)
#1028 ADD(EN: #1026.out, #1027, filterTotalAmountFT0102)
#1029 filterTotalAmountFT0102 <= #1028
#1030 NOT(DD6_DI.21)
#1031 alarmFS020101 <= #1030
#1032 NOT(DD9_DI.13)
#1033 alarmZDE0210power <= #1032
#1034 NOT(DD1_DI5)
#1035 alarmRKF <= #1034
#1036 NOT(DD9_DI.30)
#1037 alarmZDE0301power <= #1036
#1038 NOT(DD9_DI.31)
#1039 alarmZDE0302power <= #1038
#1040 MOVE(EN: filterTotalAmountReset, 0)
#1041 filterTotalAmountFT0102 <= #1040
#1042 SUB(filterValueToRegen, filterTotalAmountFT0102)
#1043 volumeToRegen <= #1042
#1044 GE(filterTotalAmountFT0102, filterValueToRegen)
#1045 MACRO управление промывкой фильтра ФС02.01.01(pin 1 "сигнал на промывку": #1044, pin 2 "авария фильтра": DD6_DI.21, pin 3 "подтверждение промывки": DD6_DI.20, pin 4 "сброс аварий": alarmReset, pin 5 "начать очередь снова": filterStartNewQueue, pin 6 "ЗДЭ02.01 открыта": DD7_DI.16, pin 7 "ЗДЭ02.01 закрыта": DD7_DI.17, pin 8 "ЗДЭ02.07 открыта": DD7_DI.28, pin 9 "ЗДЭ02.07 закрыта": DD7_DI.29, pin 10 "время движения ЗДЭ": timeToOpenCloseValve, pin 11 "авария питания ЗДЭ02.01": DD9_DI.4, pin 12 "авария питания ЗДЭ02.07": DD9_DI.10)
	(* <- выход использовать в / последнем фильтре для / начала очереди заново *)
	(* если открыт = промывка *)
	(* если открыт = фильтрация *)
	out 1 "следующий в очереди" <= #1048.output
	out 2 "промыть ФС02.01.01" <= #1047
	#1046 ZD0201:SimpleValve(inputOpen: NOT #1047, inputClose: #1047, statusOpen: pin 6, statusClose: pin 7, reset: pin 4, timeToOpenClose: pin 10)
	out 6 "открыть ЗДЭ02.01" <= #1046.outputOpen
	out 7 "закрыть ЗДЭ02.01" <= #1046.outputClose
	out 8 "авария открытия ЗДЭ02.01" <= #1046.errorToOpen
	#1047 OR(panTestValvesFS020101, #1048.regenFilterOUT)
	out 9 "авария закрытия ЗДЭ02.01" <= #1046.errorToClose
	#1048 FS020101manager:FilterQueueManager(input: pin 1, filterAlarm: #1049, regenFilterStatus: pin 3, alarmReset: pin 4, startNextLoop: pin 5)
	#1049 OR(alarmZD020107, pin 2, pin 11, pin 12)
	out 3 "ФС02.01.01 промыт" <= #1048.regenerated
	out 4 "не удалось промыть" <= #1048.failToRegen
	#1050 OR(#1046.errorToOpen, #1046.errorToClose, #1052.errorToOpen, #1052.errorToClose)
	#1051 alarmZD020107 <= #1050
	out 5 "сброс счетчика" <= #1048.counterReset
	#1052 ZD0207:SimpleValve(inputOpen: #1047, inputClose: NOT #1047, statusOpen: pin 8, statusClose: pin 9, reset: pin 4, timeToOpenClose: pin 10)
	out 10 "открыть ЗДЭ02.07" <= #1052.outputOpen
	out 11 "закрыть ЗДЭ02.07" <= #1052.outputClose
	out 12 "авария открытия ЗДЭ02.07" <= #1052.errorToOpen
	out 13 "авария закрытия ЗДЭ02.07" <= #1052.errorToClose
END_MACRO
#1053 DD2_DO.4 <= #1045.out 2
#1054 regeneratedFS020101 <= #1045.out 3
#1055 filterFailToRegen020101 <= #1045.out 4
#1056 filterTotalAmountReset <= #1045.out 5
#1057 DD2_DO.16 <= #1045.out 6
#1058 DD2_DO.17 <= #1045.out 7
#1059 errorToOpenZD0201 <= #1045.out 8
#1060 errorToCloseZD0201 <= #1045.out 9
#1061 DD2_DO.28 <= #1045.out 10
#1062 DD2_DO.29 <= #1045.out 11
#1063 errorToOpenZD0207 <= #1045.out 12
#1064 errorToCloseZD0207 <= #1045.out 13
#1065 MACRO управление промывкой фильтра ФС02.01.02(pin 1 "сигнал на промывку": #1045.out 1, pin 2 "авария фильтра": DD6_DI.23, pin 3 "подтверждение промывки": DD6_DI.22, pin 4 "сброс аварий": alarmReset, pin 5 "начать очередь снова": filterStartNewQueue, pin 6 "ЗДЭ02.02 открыта": DD7_DI.18, pin 7 "ЗДЭ02.02 закрыта": DD7_DI.19, pin 8 "ЗДЭ02.08 открыта": DD7_DI.30, pin 9 "ЗДЭ02.08 закрыта": DD7_DI.31, pin 10 "время движения ЗДЭ": timeToOpenCloseValve, pin 11 "авария питания ЗДЭ02.02": DD9_DI.5, pin 12 "авария питания ЗДЭ02.08": DD9_DI.11)
	(* <- выход использовать в / последнем фильтре для / начала очереди заново *)
	(* если открыт = промывка *)
	(* если открыт = фильтрация *)
	out 1 "следующий в очереди" <= #1068.output
	out 2 "промыть ФС02.01.02" <= #1067
	#1066 ZD0202:SimpleValve(inputOpen: NOT #1067, inputClose: #1067, statusOpen: pin 6, statusClose: pin 7, reset: pin 4, timeToOpenClose: pin 10)
	out 5 "открыть ЗДЭ02.02" <= #1066.outputOpen
	out 6 "закрыть ЗДЭ02.02" <= #1066.outputClose
	out 7 "авария открытия ЗДЭ02.02" <= #1066.errorToOpen
	#1067 OR(panTestValvesFS020102, #1068.regenFilterOUT)
	out 8 "авария закрытия ЗДЭ02.02" <= #1066.errorToClose
	#1068 FS020102manager:FilterQueueManager(input: pin 1, filterAlarm: #1069, regenFilterStatus: pin 3, alarmReset: pin 4, startNextLoop: pin 5)
	#1069 OR(alarmZD020208, pin 2, pin 11, pin 12)
	#1070 OR(#1066.errorToOpen, #1066.errorToClose, #1072.errorToOpen, #1072.errorToClose)
	#1071 alarmZD020208 <= #1070
	out 3 "ФС02.01.02 промыт" <= #1068.regenerated
	out 4 "не удалось промыть" <= #1068.failToRegen
	#1072 ZD0208:SimpleValve(inputOpen: #1067, inputClose: NOT #1067, statusOpen: pin 8, statusClose: pin 9, reset: pin 4, timeToOpenClose: pin 10)
	out 9 "открыть ЗДЭ02.08" <= #1072.outputOpen
	out 10 "закрыть ЗДЭ02.08" <= #1072.outputClose
	out 11 "авария открытия ЗДЭ02.08" <= #1072.errorToOpen
	out 12 "авария закрытия ЗДЭ02.08" <= #1072.errorToClose
END_MACRO
#1073 DD2_DO.5 <= #1065.out 2
#1074 regeneratedFS020102 <= #1065.out 3
#1075 filterFailToRegen020102 <= #1065.out 4
#1076 DD2_DO.18 <= #1065.out 5
#1077 DD2_DO.19 <= #1065.out 6
#1078 errorToOpenZD0202 <= #1065.out 7
#1079 errorToCloseZD0202 <= #1065.out 8
#1080 DD2_DO.30 <= #1065.out 9
#1081 DD2_DO.31 <= #1065.out 10
#1082 errorToOpenZD0208 <= #1065.out 11
#1083 errorToCloseZD0208 <= #1065.out 12
#1084 MACRO управление промывкой фильтра ФС02.01.03(pin 1 "сигнал на промывку": #1065.out 1, pin 2 "авария фильтра": DD6_DI.25, pin 3 "подтверждение промывки": DD6_DI.24, pin 4 "сброс аварий": alarmReset, pin 5 "начать очередь снова": filterStartNewQueue, pin 6 "ЗДЭ02.03 открыта": DD7_DI.20, pin 7 "ЗДЭ02.03 закрыта": DD7_DI.21, pin 8 "ЗДЭ02.09 открыта": DD8_DI.0, pin 9 "ЗДЭ02.09 закрыта": DD8_DI.1, pin 10 "время движения ЗДЭ": timeToOpenCloseValve, pin 11 "авария питания ЗДЭ02.03": DD9_DI.6, pin 12 "авария питания ЗДЭ02.09": DD9_DI.12)
	(* <- выход использовать в / последнем фильтре для / начала очереди заново *)
	(* если открыт = промывка *)
	(* если открыт = фильтрация *)
	out 1 "следующий в очереди" <= #1087.output
	out 2 "промыть ФС02.01.03" <= #1086
	#1085 ZD0203:SimpleValve(inputOpen: NOT #1086, inputClose: #1086, statusOpen: pin 6, statusClose: pin 7, reset: pin 4, timeToOpenClose: pin 10)
	out 5 "открыть ЗДЭ02.03" <= #1085.outputOpen
	out 6 "закрыть ЗДЭ02.03" <= #1085.outputClose
	out 7 "авария открытия ЗДЭ02.03" <= #1085.errorToOpen
	#1086 OR(panTestValvesFS020103, #1087.regenFilterOUT)
	out 8 "авария закрытия ЗДЭ02.03" <= #1085.errorToClose
	#1087 FS020103manager:FilterQueueManager(input: pin 1, filterAlarm: #1088, regenFilterStatus: pin 3, alarmReset: pin 4, startNextLoop: pin 5)
	#1088 OR(alarmZD020309, pin 2, pin 11, pin 12)
	#1089 OR(#1085.errorToOpen, #1085.errorToClose, #1091.errorToOpen, #1091.errorToClose)
	#1090 alarmZD020309 <= #1089
	out 3 "ФС02.01.03 промыт" <= #1087.regenerated
	out 4 "не удалось промыть" <= #1087.failToRegen
	#1091 ZD0209:SimpleValve(inputOpen: #1086, inputClose: NOT #1086, statusOpen: pin 8, statusClose: pin 9, reset: pin 4, timeToOpenClose: pin 10)
	out 9 "открыть ЗДЭ02.09" <= #1091.outputOpen
	out 10 "закрыть ЗДЭ02.09" <= #1091.outputClose
	out 11 "авария открытия ЗДЭ02.09" <= #1091.errorToOpen
	out 12 "авария закрытия ЗДЭ02.09" <= #1091.errorToClose
END_MACRO
#1092 DD2_DO.6 <= #1084.out 2
#1093 regeneratedFS020103 <= #1084.out 3
#1094 filterFailToRegen020103 <= #1084.out 4
#1095 DD2_DO.20 <= #1084.out 5
#1096 DD2_DO.21 <= #1084.out 6
#1097 errorToOpenZD0203 <= #1084.out 7
#1098 errorToCloseZD0203 <= #1084.out 8
#1099 DD3_DO.0 <= #1084.out 9
#1100 DD3_DO.1 <= #1084.out 10
#1101 errorToOpenZD0209 <= #1084.out 11
#1102 errorToCloseZD0209 <= #1084.out 12
#1103 MACRO управление промывкой фильтра ФС02.01.04(pin 1 "сигнал на промывку": #1084.out 1, pin 2 "авария фильтра": DD6_DI.27, pin 3 "подтверждение промывки": DD6_DI.26, pin 4 "сброс аварий": alarmReset, pin 5 "начать очередь снова": filterStartNewQueue, pin 6 "ЗДЭ02.04 открыта": DD7_DI.22, pin 7 "ЗДЭ02.04 закрыта": DD7_DI.23, pin 8 "ЗДЭ02.10 открыта": DD8_DI.2, pin 9 "ЗДЭ02.10 закрыта": DD8_DI.3, pin 10 "время движения ЗДЭ": timeToOpenCloseValve, pin 11 "авария питания ЗДЭ02.04": DD9_DI.7, pin 12 "авария питания ЗДЭ02.10": DD9_DI.13)
	(* <- выход использовать в / последнем фильтре для / начала очереди заново *)
	(* если открыт = промывка *)
	(* если открыт = фильтрация *)
	out 1 "следующий в очереди" <= #1106.output
	out 2 "промыть ФС02.01.04" <= #1105
	#1104 ZD0204:SimpleValve(inputOpen: NOT #1105, inputClose: #1105, statusOpen: pin 6, statusClose: pin 7, reset: pin 4, timeToOpenClose: pin 10)
	out 5 "открыть ЗДЭ02.04" <= #1104.outputOpen
	out 6 "закрыть ЗДЭ02.04" <= #1104.outputClose
	out 7 "авария открытия ЗДЭ02.04" <= #1104.errorToOpen
	#1105 OR(panTestValvesFS020104, #1106.regenFilterOUT)
	out 8 "авария закрытия ЗДЭ02.04" <= #1104.errorToClose
	#1106 FS020104manager:FilterQueueManager(input: pin 1, filterAlarm: #1107, regenFilterStatus: pin 3, alarmReset: pin 4, startNextLoop: pin 5)
	#1107 OR(alarmZD020410, pin 2, pin 11, pin 12)
	#1108 OR(#1104.errorToOpen, #1104.errorToClose, #1110.errorToOpen, #1110.errorToClose)
	#1109 alarmZD020410 <= #1108
	out 3 "ФС02.01.04 промыт" <= #1106.regenerated
	out 4 "не удалось промыть" <= #1106.failToRegen
	#1110 ZD0210:SimpleValve(inputOpen: #1105, inputClose: NOT #1105, statusOpen: pin 8, statusClose: pin 9, reset: pin 4, timeToOpenClose: pin 10)
	out 9 "открыть ЗДЭ02.10" <= #1110.outputOpen
	out 10 "закрыть ЗДЭ02.10" <= #1110.outputClose
	out 11 "авария открытия ЗДЭ02.10" <= #1110.errorToOpen
	out 12 "авария закрытия ЗДЭ02.10" <= #1110.errorToClose
END_MACRO
#1111 DD2_DO.7 <= #1103.out 2
#1112 regeneratedFS020104 <= #1103.out 3
#1113 filterFailToRegen020104 <= #1103.out 4
#1114 DD2_DO.22 <= #1103.out 5
#1115 DD2_DO.23 <= #1103.out 6
#1116 errorToOpenZD0204 <= #1103.out 7
#1117 errorToCloseZD0204 <= #1103.out 8
#1118 DD3_DO.2 <= #1103.out 9
#1119 DD3_DO.3 <= #1103.out 10
#1120 errorToOpenZD0210 <= #1103.out 11
#1121 errorToCloseZD0210 <= #1103.out 12
#1122 MACRO управление промывкой фильтра ФС02.01.05(pin 1 "сигнал на промывку": #1103.out 1, pin 2 "авария фильтра": DD6_DI.29, pin 3 "подтверждение промывки": DD6_DI.28, pin 4 "сброс аварий": alarmReset, pin 5 "начать очередь снова": filterStartNewQueue, pin 6 "ЗДЭ02.05 открыта": DD7_DI.24, pin 7 "ЗДЭ02.05 закрыта": DD7_DI.25, pin 8 "ЗДЭ02.11 открыта": DD8_DI.4, pin 9 "ЗДЭ02.11 закрыта": DD8_DI.5, pin 10 "время движения ЗДЭ": timeToOpenCloseValve, pin 11 "авария питания ЗДЭ02.05": DD9_DI.8, pin 12 "авария питания ЗДЭ02.11": DD9_DI.14)
	(* <- выход использовать в / последнем фильтре для / начала очереди заново *)
	(* если открыт = промывка *)
	(* если открыт = фильтрация *)
	out 1 "следующий в очереди" <= #1125.output
	out 2 "промыть ФС02.01.05" <= #1124
	#1123 ZD0205:SimpleValve(inputOpen: NOT #1124, inputClose: #1124, statusOpen: pin 6, statusClose: pin 7, reset: pin 4, timeToOpenClose: pin 10)
	out 5 "открыть ЗДЭ02.05" <= #1123.outputOpen
	out 6 "закрыть ЗДЭ02.05" <= #1123.outputClose
	out 7 "авария открытия ЗДЭ02.05" <= #1123.errorToOpen
	#1124 OR(panTestValvesFS020105, #1125.regenFilterOUT)
	out 8 "авария закрытия ЗДЭ02.05" <= #1123.errorToClose
	#1125 FS020105manager:FilterQueueManager(input: pin 1, filterAlarm: #1126, regenFilterStatus: pin 3, alarmReset: pin 4, startNextLoop: pin 5)
	#1126 OR(alarmZD020511, pin 2, pin 11, pin 12)
	#1127 OR(#1123.errorToOpen, #1123.errorToClose, #1129.errorToOpen, #1129.errorToClose)
	#1128 alarmZD020511 <= #1127
	out 3 "ФС02.01.05 промыт" <= #1125.regenerated
	out 4 "не удалось промыть" <= #1125.failToRegen
	#1129 ZD0211:SimpleValve(inputOpen: #1124, inputClose: NOT #1124, statusOpen: pin 8, statusClose: pin 9, reset: pin 4, timeToOpenClose: pin 10)
	out 9 "открыть ЗДЭ02.11" <= #1129.outputOpen
	out 10 "закрыть ЗДЭ02.11" <= #1129.outputClose
	out 11 "авария открытия ЗДЭ02.11" <= #1129.errorToOpen
	out 12 "авария закрытия ЗДЭ02.11" <= #1129.errorToClose
END_MACRO
#1130 DD2_DO.8 <= #1122.out 2
#1131 regeneratedFS020105 <= #1122.out 3
#1132 filterFailToRegen020105 <= #1122.out 4
#1133 DD2_DO.24 <= #1122.out 5
#1134 DD2_DO.25 <= #1122.out 6
#1135 errorToOpenZD0205 <= #1122.out 7
#1136 errorToCloseZD0205 <= #1122.out 8
#1137 DD3_DO.4 <= #1122.out 9
#1138 DD3_DO.5 <= #1122.out 10
#1139 errorToOpenZD0211 <= #1122.out 11
#1140 errorToCloseZD0211 <= #1122.out 12
#1141 MACRO управление промывкой фильтра ФС02.01.06(pin 1 "сигнал на промывку": #1122.out 1, pin 2 "авария фильтра": DD6_DI.31, pin 3 "подтверждение промывки": DD6_DI.30, pin 4 "сброс аварий": alarmReset, pin 5 "начать очередь снова": filterStartNewQueue, pin 6 "ЗДЭ02.06 открыта": DD7_DI.26, pin 7 "ЗДЭ02.06 закрыта": DD7_DI.27, pin 8 "ЗДЭ02.12 открыта": DD8_DI.6, pin 9 "ЗДЭ02.12 закрыта": DD8_DI.7, pin 10 "время движения ЗДЭ": timeToOpenCloseValve, pin 11 "авария питания ЗДЭ02.06": DD9_DI.9, pin 12 "авария питания ЗДЭ02.12": DD9_DI.15)
	(* <- выход использовать в / последнем фильтре для / начала очереди заново *)
	(* если открыт = промывка *)
	(* если открыт = фильтрация *)
	out 1 "следующий в очереди" <= #1144.output
	out 2 "промыть ФС02.01.06" <= #1143
	#1142 ZD0206:SimpleValve(inputOpen: NOT #1143, inputClose: #1143, statusOpen: pin 6, statusClose: pin 7, reset: pin 4, timeToOpenClose: pin 10)
	out 5 "открыть ЗДЭ02.06" <= #1142.outputOpen
	out 6 "закрыть ЗДЭ02.06" <= #1142.outputClose
	out 7 "авария открытия ЗДЭ02.06" <= #1142.errorToOpen
	#1143 OR(panTestValvesFS020106, #1144.regenFilterOUT)
	out 8 "авария закрытия ЗДЭ02.06" <= #1142.errorToClose
	#1144 FS020106manager:FilterQueueManager(input: pin 1, filterAlarm: #1145, regenFilterStatus: pin 3, alarmReset: pin 4, startNextLoop: pin 5)
	#1145 OR(alarmZD020612, pin 2, pin 11, pin 12)
	#1146 OR(#1142.errorToOpen, #1142.errorToClose, #1148.errorToOpen, #1148.errorToClose)
	#1147 alarmZD020612 <= #1146
	out 3 "ФС02.01.06 промыт" <= #1144.regenerated
	out 4 "не удалось промыть" <= #1144.failToRegen
	#1148 ZD0212:SimpleValve(inputOpen: #1143, inputClose: NOT #1143, statusOpen: pin 8, statusClose: pin 9, reset: pin 4, timeToOpenClose: pin 10)
	out 9 "открыть ЗДЭ02.12" <= #1148.outputOpen
	out 10 "закрыть ЗДЭ02.12" <= #1148.outputClose
	out 11 "авария открытия ЗДЭ02.12" <= #1148.errorToOpen
	out 12 "авария закрытия ЗДЭ02.12" <= #1148.errorToClose
END_MACRO
#1149 DD2_DO.9 <= #1141.out 2
#1150 regeneratedFS020106 <= #1141.out 3
#1151 filterFailToRegen020106 <= #1141.out 4
#1152 DD2_DO.26 <= #1141.out 5
#1153 DD2_DO.27 <= #1141.out 6
#1154 errorToOpenZD0206 <= #1141.out 7
#1155 errorToCloseZD0206 <= #1141.out 8
#1156 DD3_DO.6 <= #1141.out 9
#1157 DD3_DO.7 <= #1141.out 10
#1158 errorToOpenZD0212 <= #1141.out 11
#1159 errorToCloseZD0212 <= #1141.out 12
#1160 MACRO управление промывкой фильтра ФС02.02.01(pin 1 "сигнал на промывку": #1141.out 1, pin 2 "авария фильтра": DD7_DI.1, pin 3 "подтверждение промывки": DD7_DI.0, pin 4 "сброс аварий": alarmReset, pin 5 "начать очередь снова": filterStartNewQueue, pin 6 "ЗДЭ02.13 открыта": DD8_DI.8, pin 7 "ЗДЭ02.13 закрыта": DD8_DI.9, pin 8 "ЗДЭ02.19 открыта": DD8_DI.20, pin 9 "ЗДЭ02.19 закрыта": DD8_DI.21, pin 10 "время движения ЗДЭ": timeToOpenCloseValve, pin 11 "авария питания ЗДЭ02.13": DD9_DI.16, pin 12 "авария питания ЗДЭ02.19": DD9_DI.22)
	(* <- выход использовать в / последнем фильтре для / начала очереди заново *)
	(* если открыт = промывка *)
	(* если открыт = фильтрация *)
	out 1 "следующий в очереди" <= #1163.output
	out 2 "промыть ФС02.02.01" <= #1162
